(* IEC 61131-3 sources: Yaha/Documentation/Infomaterial/OSCAT/pcworx_basic_333/module_export (part 8) *)

(* ---- MS_TO_KMH.ST ---- *)
(*@PROPERTIES_EX@
TYPE: POU
LOCALE: 0
IEC_LANGUAGE: ST
PLC_TYPE: independent
PROC_TYPE: independent
GROUP: ENGINEERING.CONVERSION
*)
(*@KEY@:DESCRIPTION*)
version 1.0	4 Feb 2007
programmer 	hugo
tested by	tobias

this function converts velocities from Meters / Second to Kilometers / hour.
(*@KEY@:END_DESCRIPTION*)
FUNCTION MS_TO_KMH:REAL

(*Group:Default*)

VAR_INPUT
	MS :	REAL;
END_VAR

(*@KEY@: WORKSHEET
NAME: MS_TO_KMH
IEC_LANGUAGE: ST
*)
MS_TO_KMH := ms * 3.6;
(*@KEY@: END_WORKSHEET *)
END_FUNCTION

(* ---- MUL_ADD.ST ---- *)
(*@PROPERTIES_EX@
TYPE: POU
LOCALE: 0
IEC_LANGUAGE: ST
PLC_TYPE: independent
PROC_TYPE: independent
GROUP: MATHEMATICAL.MATHE
*)
(*@KEY@:DESCRIPTION*)
version 1.1	11 nov 2007
programmer 	hugo
tested by	tobias

this function multiplies an input X with K and adds Offset O to the result.
(*@KEY@:END_DESCRIPTION*)
FUNCTION MUL_ADD:REAL

(*Group:Default*)

VAR_INPUT
	X :	REAL;
	K :	REAL;
	O :	REAL;
END_VAR

(*@KEY@: WORKSHEET
NAME: MUL_ADD
IEC_LANGUAGE: ST
*)
MUL_ADD := X * K + O;
(*@KEY@: END_WORKSHEET *)
END_FUNCTION

(* ---- MULTI_IN.ST ---- *)
(*@PROPERTIES_EX@
TYPE: POU
LOCALE: 0
IEC_LANGUAGE: ST
PLC_TYPE: independent
PROC_TYPE: independent
GROUP: ENGINEERING.SENSOR
*)
(*@KEY@:DESCRIPTION*)
version 1.4	18. jul. 2009
programmer 	oscat
tested by	oscat

multi_in is a signal conditioning function which can be configured in 8 different ways.
it is used to read multiple sensors for the same value and protect the user from broken sensors or invalid data from sensors.

multi_in can be configured in different ways:
	mode = 0 means the the avg of the 3 inputs is used, this mode is the default mode.
	mode = 1 means in_1 is used.
	mode = 2 means in_2 is used.
	mode = 3 means in_3 is used.
	mode = 4 means default is used.
	mode = 5 means the lowest of the 3 external temperatures is used.
	mode = 6 means the higest externnal temperature is used.
	mode = 7 means the midlle input is used, if there are only two working, the lowest input is used.
	mode > 7 ,eans output is 0 at all times.
	in any config mode, an input higher then in_max or lower then in_min is ignored to prevent values from broken sensors or wires.
	if all inputs are higher then in_max or lower then in_min, a default value (default) is used.

(*@KEY@:END_DESCRIPTION*)
FUNCTION MULTI_IN:REAL

(*Group:Default*)

VAR_INPUT
	IN_1 :	REAL;
	IN_2 :	REAL;
	IN_3 :	REAL;
	DEFAULT :	REAL;
	IN_MIN :	REAL;
	IN_MAX :	REAL;
	MODE :	BYTE;
END_VAR

VAR
	count :	INT;
	F1 :	BOOL;
	F2 :	BOOL;
	F3 :	BOOL;
END_VAR

(*@KEY@: WORKSHEET
NAME: MULTI_IN
IEC_LANGUAGE: ST
*)
F1 :=  in_1 > in_min AND in_1 < in_max;
F2 :=  in_2 > in_min AND in_2 < in_max;
F3 :=  in_3 > in_min AND in_3 < in_max;

CASE _BYTE_TO_INT(mode) OF
0:	count := 0;
	IF F1 THEN
		count := count + 1;
		MULTI_IN := in_1;
	ELSE
		MULTI_IN := 0.0;
	END_IF;
	IF F2 THEN
		count := count + 1;
		MULTI_IN := MULTI_IN + in_2;
	END_IF;
	IF F3 THEN
		count := count + 1;
		MULTI_IN := MULTI_IN + in_3;
	END_IF;
	MULTI_IN := SEL_REAL(count = 0, MULTI_IN / INT_TO_REAL(count), default);

1:	MULTI_IN := SEL_REAL(F1, default, IN_1);

2:	MULTI_IN := SEL_REAL(F2, default, IN_2);

3:	MULTI_IN := SEL_REAL(F3, default, IN_3);

4:	MULTI_IN := default;

5:	MULTI_IN := SEL_REAL(F1, in_max, IN_1);
	IF F2 AND in_2 < MULTI_IN THEN MULTI_IN := in_2; END_IF;
	IF F3 AND in_3 < MULTI_IN THEN MULTI_IN := in_3; END_IF;
	IF MULTI_IN = in_max THEN MULTI_IN := default; END_IF;

6:	MULTI_IN := SEL_REAL(F1, in_min, IN_1);
	IF F2 AND in_2 > MULTI_IN THEN MULTI_IN := in_2; END_IF;
	IF F3 AND in_3 > MULTI_IN THEN MULTI_IN := in_3; END_IF;
	IF MULTI_IN = in_min THEN MULTI_IN := default; END_IF;

7:	IF F1 AND F2 AND F3 THEN MULTI_IN := MID3(in_1, in_2, in_3);
	ELSIF F1 AND F2 THEN MULTI_IN := MIN(in_1, in_2);
	ELSIF F1 AND F3 THEN MULTI_IN := MIN(in_1, in_3);
	ELSIF F2 AND F3 THEN MULTI_IN := MIN(in_2, in_3);
	ELSIF F1 THEN MULTI_IN := in_1;
	ELSIF F2 THEN MULTI_IN := in_2;
	ELSIF F3 THEN MULTI_IN := in_3;
	ELSE MULTI_IN := default;
	END_IF;

END_CASE;

(*
hm 1.1.2007		rev 1.1
	changed midr to mid3 function

hm	14. 10. 2008	rev 1.2
	corrected an error for in_3 overrange detection
	improved performance

hm	11. mar. 2009	rev 1.3
	changed real constants to use dot syntax

hm	18. jul. 2009	rev 1.4
	improved performance
*)

(*@KEY@: END_WORKSHEET *)
END_FUNCTION

(* ---- MULTIME.ST ---- *)
(*@PROPERTIES_EX@
TYPE: POU
LOCALE: 0
IEC_LANGUAGE: ST
PLC_TYPE: independent
PROC_TYPE: independent
GROUP: TIME_DATE
*)
(*@KEY@:DESCRIPTION*)
version 1.1	14 mar 2008
programmer 	hugo
tested by	tobias

multiplies a time by a real number and returns a time
(*@KEY@:END_DESCRIPTION*)
FUNCTION MULTIME:TIME

(*Group:Default*)

VAR_INPUT
	T :	TIME;
	M :	REAL;
END_VAR

(*@KEY@: WORKSHEET
NAME: MULTIME
IEC_LANGUAGE: ST
*)
multime := DWORD_TO_TIME(_REAL_TO_DWORD(_DWORD_TO_REAL(TIME_TO_DWORD(t))*M));

(* revision history
hm		2. oct 2006	rev 1.0
	original version

hm		14. mar 2008	rev 1.1
	rounded the result after the last digit

*)
(*@KEY@: END_WORKSHEET *)
END_FUNCTION

(* ---- MUX_2.ST ---- *)
(*@PROPERTIES_EX@
TYPE: POU
LOCALE: 0
IEC_LANGUAGE: ST
PLC_TYPE: independent
PROC_TYPE: independent
GROUP: LOGIC.GATE_LOGIC
*)
(*@KEY@:DESCRIPTION*)
version 1.2	16. oct. 2008
programmer 	hugo
tested BY	oscat

dual input multiplexer
depending on the value of A0, D0 or D1 will be switched to the Output
(*@KEY@:END_DESCRIPTION*)
FUNCTION MUX_2:BOOL

(*Group:Default*)

VAR_INPUT
	D0 :	BOOL;
	D1 :	BOOL;
	A0 :	BOOL;
END_VAR

(*@KEY@: WORKSHEET
NAME: MUX_2
IEC_LANGUAGE: ST
*)
MUX_2 := SEL(A0, D0, D1);

(*
revision history:
hm	5.10.2006		rev 1.1
	changed to ST Langage for better portability.

hm	16. oct. 2008	rev 1.2
	improved performance

*)
(*@KEY@: END_WORKSHEET *)
END_FUNCTION

(* ---- MUX_4.ST ---- *)
(*@PROPERTIES_EX@
TYPE: POU
LOCALE: 0
IEC_LANGUAGE: ST
PLC_TYPE: independent
PROC_TYPE: independent
GROUP: LOGIC.GATE_LOGIC
*)
(*@KEY@:DESCRIPTION*)
version 1.2	16. oct. 2008
programmer 	hugo
tested BY	oscat

quad input multiplexer
depending on the value of A0 and A1, one of the 4 inputs will be switched to the Output
(*@KEY@:END_DESCRIPTION*)
FUNCTION MUX_4:BOOL

(*Group:Default*)

VAR_INPUT
	D0 :	BOOL;
	D1 :	BOOL;
	D2 :	BOOL;
	D3 :	BOOL;
	A0 :	BOOL;
	A1 :	BOOL;
END_VAR

(*@KEY@: WORKSHEET
NAME: MUX_4
IEC_LANGUAGE: ST
*)
IF A1 THEN
	MUX_4 := SEL(A0, D2, D3);
ELSE
	MUX_4 := SEL(A0, D0, D1);
END_IF;

(*
revision history:
hm 	5.10.2006		rev 1.1
	rewritten to ST for better portability

hm	16. oct. 2008	rev 1.2
	improved performance

*)
(*@KEY@: END_WORKSHEET *)
END_FUNCTION

(* ---- MUX_R2.ST ---- *)
(*@PROPERTIES_EX@
TYPE: POU
LOCALE: 0
IEC_LANGUAGE: ST
PLC_TYPE: independent
PROC_TYPE: independent
GROUP: ENGINEERING.SIGNAL_PROCESSING
*)
(*@KEY@:DESCRIPTION*)
version 1.1	16. oct. 2008
programmer 	oscat
tested by	oscat

MUX_R2 is an analog Multiplexer.
one of 2 real inputs are selected and put through to out.
The Adress input A selects between 2 Real inputs IN0 and IN1, A=0 > In0, A=1 > in1.
(*@KEY@:END_DESCRIPTION*)
FUNCTION MUX_R2:REAL

(*Group:Default*)

VAR_INPUT
	IN0 :	REAL;
	IN1 :	REAL;
	A :	BOOL;
END_VAR

(*@KEY@: WORKSHEET
NAME: MUX_R2
IEC_LANGUAGE: ST
*)
MUX_R2 := SEL(A, IN0, IN1);

(* revision history
hm	19. jan. 2007	rev 1.0
	original version

hm	16. oct. 2008	rev 1.1
	improved performance
*)
(*@KEY@: END_WORKSHEET *)
END_FUNCTION

(* ---- MUX_R4.ST ---- *)
(*@PROPERTIES_EX@
TYPE: POU
LOCALE: 0
IEC_LANGUAGE: ST
PLC_TYPE: independent
PROC_TYPE: independent
GROUP: ENGINEERING.SIGNAL_PROCESSING
*)
(*@KEY@:DESCRIPTION*)
version 1.1	16. oct. 2008
programmer 	oscat
tested by	oscat

MUX_R4 is an analog Multiplexer.
one of 4 real inputs are selected and put through to out.
The Adress input A0 and A1 selects between the 4 Real inputs IN0.. IN1.
(*@KEY@:END_DESCRIPTION*)
FUNCTION MUX_R4:REAL

(*Group:Default*)

VAR_INPUT
	IN0 :	REAL;
	IN1 :	REAL;
	IN2 :	REAL;
	IN3 :	REAL;
	A0 :	BOOL;
	A1 :	BOOL;
END_VAR

(*@KEY@: WORKSHEET
NAME: MUX_R4
IEC_LANGUAGE: ST
*)
IF A1 THEN
	MUX_R4 := SEL(A0, IN2, IN3);
ELSE
	MUX_R4 := SEL(A0, IN0, IN1);
END_IF;

(* revision history
hm	19. jan 2007	rev 1.0
	original version

hm	16. oct. 2008	rev 1.1
	improved performance
*)
(*@KEY@: END_WORKSHEET *)
END_FUNCTION

(* ---- NEGX.ST ---- *)
(*@PROPERTIES_EX@
TYPE: POU
LOCALE: 0
IEC_LANGUAGE: ST
PLC_TYPE: independent
PROC_TYPE: independent
GROUP: MATHEMATICAL.MATHE
*)
(*@KEY@:DESCRIPTION*)
version 1.0	26. oct. 2008
programmer 	hugo
tested by	tobias

This function returns -X
(*@KEY@:END_DESCRIPTION*)
FUNCTION NEGX:REAL

(*Group:Default*)

VAR_INPUT
	X :	REAL;
END_VAR

(*@KEY@: WORKSHEET
NAME: NEGX
IEC_LANGUAGE: ST
*)
NEGX := -X;

(* revision history
hm	26. oct. 2008	rev 1.0
	original version

*)
(*@KEY@: END_WORKSHEET *)
END_FUNCTION

(* ---- OFFSET.ST ---- *)
(*@PROPERTIES_EX@
TYPE: POU
LOCALE: 0
IEC_LANGUAGE: ST
PLC_TYPE: independent
PROC_TYPE: independent
GROUP: ENGINEERING.SIGNAL_PROCESSING
*)
(*@KEY@:DESCRIPTION*)
version 1.0	12 jan 2007
programmer 	oscat
tested by	tobias

The Function offset adds offsets to an analog signal depending on digital inputs.
all selected offsets are added at the same time.
with the input D a default value instead of the input X can be used.
(*@KEY@:END_DESCRIPTION*)
FUNCTION OFFSET:REAL

(*Group:Default*)

VAR_INPUT
	X :	REAL;
	O1 :	BOOL;
	O2 :	BOOL;
	O3 :	BOOL;
	O4 :	BOOL;
	D :	BOOL;
	OFFSET_1 :	REAL;
	OFFSET_2 :	REAL;
	OFFSET_3 :	REAL;
	OFFSET_4 :	REAL;
	DEFAULT :	REAL;
END_VAR

(*@KEY@: WORKSHEET
NAME: OFFSET
IEC_LANGUAGE: ST
*)
IF D THEN Offset := default; ELSE Offset := X; END_IF;
IF O1 THEN Offset := Offset + offset_1; END_IF;
IF O2 THEN Offset := Offset + offset_2; END_IF;
IF O3 THEN Offset := Offset + offset_3; END_IF;
IF O4 THEN Offset := Offset + offset_4; END_IF;
(*@KEY@: END_WORKSHEET *)
END_FUNCTION

(* ---- OFFSET2.ST ---- *)
(*@PROPERTIES_EX@
TYPE: POU
LOCALE: 0
IEC_LANGUAGE: ST
PLC_TYPE: independent
PROC_TYPE: independent
GROUP: ENGINEERING.SIGNAL_PROCESSING
*)
(*@KEY@:DESCRIPTION*)
version 1.0	12 jan 2007
programmer 	oscat
tested by	tobias

The Function offset adds offsets to an analog signal depending on digital inputs.
one offset can be added at the same time, if more then one input is true, the one with the highest number (o1 .. o4) will be used.
The input D will select a default value instead of X for input.
(*@KEY@:END_DESCRIPTION*)
FUNCTION OFFSET2:REAL

(*Group:Default*)

VAR_INPUT
	X :	REAL;
	O1 :	BOOL;
	O2 :	BOOL;
	O3 :	BOOL;
	O4 :	BOOL;
	D :	BOOL;
	OFFSET_1 :	REAL;
	OFFSET_2 :	REAL;
	OFFSET_3 :	REAL;
	OFFSET_4 :	REAL;
	DEFAULT :	REAL;
END_VAR

(*@KEY@: WORKSHEET
NAME: OFFSET2
IEC_LANGUAGE: ST
*)
IF D THEN Offset2 := default; ELSE Offset2 := X; END_IF;
IF O4 THEN Offset2 := Offset2 + offset_4;
ELSIF O3 THEN Offset2 := Offset2 + offset_3;
ELSIF O2 THEN Offset2 := Offset2 + offset_2;
ELSIF O1 THEN Offset2 := Offset2 + offset_1;
END_IF;
(*@KEY@: END_WORKSHEET *)
END_FUNCTION

(* ---- OM_TO_F.ST ---- *)
(*@PROPERTIES_EX@
TYPE: POU
LOCALE: 0
IEC_LANGUAGE: ST
PLC_TYPE: independent
PROC_TYPE: independent
GROUP: ENGINEERING.CONVERSION
*)
(*@KEY@:DESCRIPTION*)
version 1.1	18. oct. 2008
programmer 	hugo
tested by		tobias

this function converts Omega F to frequency
F = OM / (2*PI)
(*@KEY@:END_DESCRIPTION*)
FUNCTION OM_TO_F:REAL

(*Group:Default*)

VAR_INPUT
	OM :	REAL;
END_VAR

(*@KEY@: WORKSHEET
NAME: OM_TO_F
IEC_LANGUAGE: ST
*)
OM_to_F := OM / 6.283185307179586476;

(* revision history
hm	22. jan. 2007	rev 1.0
	original version

hm	18. oct. 2008	rev 1.1
	using math constants

*)
(*@KEY@: END_WORKSHEET *)
END_FUNCTION

(* ---- OSCAT_VERSION.ST ---- *)
(*@PROPERTIES_EX@
TYPE: POU
LOCALE: 0
IEC_LANGUAGE: ST
PLC_TYPE: independent
PROC_TYPE: independent
GROUP: OTHER
*)
(*@KEY@:DESCRIPTION*)
version 1.1	16 dec 2007
programmer 	hugo
tested by	tobias

oscat_version returns the version number in dword format
132 is library version 1.32
if IN = true, the release date will be returned
(*@KEY@:END_DESCRIPTION*)
FUNCTION OSCAT_VERSION:DWORD

(*Group:Default*)

VAR_INPUT
	IN :	BOOL;
END_VAR

(*@KEY@: WORKSHEET
NAME: OSCAT_VERSION
IEC_LANGUAGE: ST
*)
IF in THEN
	Oscat_version := UDINT_TO_DWORD(set_Date(2012,01,02));
ELSE
	Oscat_version := DWORD#333;
END_IF;

(* revision history
hm	6. oct 2006	rev 1.0
	original version

hm	16. dec 2007	rev 1.1
	added possibility to return date and version depending on IN.

*)
(*@KEY@: END_WORKSHEET *)
END_FUNCTION

(* ---- PARITY.ST ---- *)
(*@PROPERTIES_EX@
TYPE: POU
LOCALE: 0
IEC_LANGUAGE: ST
PLC_TYPE: independent
PROC_TYPE: independent
GROUP: LOGIC.GATE_LOGIC
*)
(*@KEY@:DESCRIPTION*)
version 1.3	18 feb 2008
programmer 	hugo
tested BY	hans

this function calculates the even parity of an input Dword
the output will be true if the amount of high bits are an odd number.
(*@KEY@:END_DESCRIPTION*)
FUNCTION PARITY:BOOL

(*Group:Default*)

VAR_INPUT
	IN :	DWORD;
END_VAR

VAR
	in2 :	DWORD;
END_VAR

(*@KEY@: WORKSHEET
NAME: PARITY
IEC_LANGUAGE: ST
*)
in2:=in;
WHILE in2 > DWORD#0 DO
	parity := parity XOR BIT_OF_DWORD(in2,0) XOR BIT_OF_DWORD(in2,1) XOR BIT_OF_DWORD(in2,2) XOR BIT_OF_DWORD(in2,3);
	in2 := SHR(in2,4);
END_WHILE;

(* code before rev 1.2
WHILE in > 0 DO
	IF in.0 THEN cnt := cnt +1; END_IF;
	in := SHR(in,1);
END_WHILE;
IF (cnt MOD 2) = 1 THEN parity := TRUE; ELSE parity := FALSE; END_IF;
*)

(* revision history

rev 1.0 hm 1 sep 2006
	original version

rev 1.1 hm 10.9.2007
	changed algorithm to improve performance

rev 1.2	hm	8 dec 2007
	changed algorithm to improve performance

rev 1.3	hm	18 feb 2008
	changed algorithm to improve performance
*)
(*@KEY@: END_WORKSHEET *)
END_FUNCTION

(* ---- PERIOD.ST ---- *)
(*@PROPERTIES_EX@
TYPE: POU
LOCALE: 0
IEC_LANGUAGE: ST
PLC_TYPE: independent
PROC_TYPE: independent
GROUP: TIME_DATE
*)
(*@KEY@:DESCRIPTION*)
version 1.3	22. mar. 2008
programmer 	hugo
tested by	tobias

PERIOD checks if a given date is between two dates (d1 and d2) d1 is the starting date and d2 the last date for the period.
the years of the dates are ignored, so the function period cheks for a time period within a year independet of the year.
(*@KEY@:END_DESCRIPTION*)
FUNCTION PERIOD:BOOL

(*Group:Default*)

VAR
	day1 :	INT;
	day2 :	INT;
	dayx :	INT;
END_VAR

VAR_INPUT
	D1 :	UDINT;
	Dx :	UDINT;
	D2 :	UDINT;
END_VAR

(*@KEY@: WORKSHEET
NAME: PERIOD
IEC_LANGUAGE: ST
*)
day1 := day_of_year(d1);
day2 := day_of_year(d2);
dayx := day_of_year(dx);
IF NOT leap_of_Date(dx) AND dayx > 58 THEN dayx := dayx + 1; END_IF;
IF NOT leap_of_Date(d1) AND day1 > 58 THEN day1 := day1 + 1; END_IF;
IF NOT leap_of_Date(d2) AND day2 > 58 THEN day2 := day2 + 1; END_IF;

IF day2 < day1 THEN
	(* the period spans over the new year *)
	period := dayx <= day2 OR dayx >= day1;
ELSE
	period := dayx >= day1 AND dayx <= day2;
END_IF;

(* code before rev 1.2
yx := year(dx);
p1 := date_add(d1,0,0,0,yx - year(d1));
p2 := date_add(d2,0,0,0,yx - year(d2));

IF p2 >= p1 THEN
	period := dx <= p2  AND dx >= p1;
ELSE
	period := dx <= p2 OR dx >= p1;
END_IF;
*)

(* revision history

hm		19. sep 2007	rev 1.0
	original version

hm		20. sep 2007	rev 1.1
	corrected a problem with leap year

hm		4. jan 2008		rev 1.2
	changed code for better performance

hm		22. mar. 2008	rev 1.3
	function would deliver wrong results when d1, d2 or dx are a leap_year

*)
(*@KEY@: END_WORKSHEET *)
END_FUNCTION

(* ---- PT_TO_F.ST ---- *)
(*@PROPERTIES_EX@
TYPE: POU
LOCALE: 0
IEC_LANGUAGE: ST
PLC_TYPE: independent
PROC_TYPE: independent
GROUP: ENGINEERING.CONVERSION
*)
(*@KEY@:DESCRIPTION*)
version 1.1	11. mar. 2009
programmer 	hugo
tested by	tobias

this function converts periode time to frequency
(*@KEY@:END_DESCRIPTION*)
FUNCTION PT_TO_F:REAL

(*Group:Default*)

VAR_INPUT
	PT :	TIME;
END_VAR

(*@KEY@: WORKSHEET
NAME: PT_TO_F
IEC_LANGUAGE: ST
*)
PT_TO_F := 1000.0 / _DWORD_TO_REAL(TIME_TO_DWORD(PT));

(*	revision history
hm	4. aug. 2006	rev 1.0
	original version

hm	11. mar. 2009	rev 1.1
	real constants updated to new systax using dot

*)
(*@KEY@: END_WORKSHEET *)
END_FUNCTION

(* ---- RAD.ST ---- *)
(*@PROPERTIES_EX@
TYPE: POU
LOCALE: 0
IEC_LANGUAGE: ST
PLC_TYPE: independent
PROC_TYPE: independent
GROUP: MATHEMATICAL.MATHE
*)
(*@KEY@:DESCRIPTION*)
version 1.2	18. oct. 2008
programmer 	hugo
tested by	tobias

this function converts Radiant to degrees
(*@KEY@:END_DESCRIPTION*)
FUNCTION RAD:REAL

(*Group:Default*)

VAR_INPUT
	DEG :	REAL;
END_VAR

(*@KEY@: WORKSHEET
NAME: RAD
IEC_LANGUAGE: ST
*)
Rad := modR(0.0174532925199433 * deg , 6.283185307179586476);

(* revision history
hm	4. aug 2006		rev 1.0
	original version

hm 	16. oct 2007	rev 1.1
	added modr statement which prohibits rad to become bigger than 2PI

hm	18. oct 2008	rev 1.2
	using math constants

*)
(*@KEY@: END_WORKSHEET *)
END_FUNCTION

(* ---- RANGE_TO_BYTE.ST ---- *)
(*@PROPERTIES_EX@
TYPE: POU
LOCALE: 0
IEC_LANGUAGE: ST
PLC_TYPE: independent
PROC_TYPE: independent
GROUP: ENGINEERING.SIGNAL_PROCESSING
*)
(*@KEY@:DESCRIPTION*)
version 1.0	9. jan 2008
programmer 	hugo
tested by		tobias

Range_to_byte converts a real value between low and high into a byte
(*@KEY@:END_DESCRIPTION*)
FUNCTION RANGE_TO_BYTE:BYTE

(*Group:Default*)

VAR_INPUT
	X :	REAL;
	LOW :	REAL;
	HIGH :	REAL;
END_VAR

(*@KEY@: WORKSHEET
NAME: RANGE_TO_BYTE
IEC_LANGUAGE: ST
*)
Range_to_Byte := REAL_TO_BYTE(TRUNC_REAL((LIMIT(low,X,high)-low) * 255.0 / (high - low)));

(* revision history
hm	9. jan 2008		rev 1.0
	original version

*)
(*@KEY@: END_WORKSHEET *)
END_FUNCTION

(* ---- RANGE_TO_WORD.ST ---- *)
(*@PROPERTIES_EX@
TYPE: POU
LOCALE: 0
IEC_LANGUAGE: ST
PLC_TYPE: independent
PROC_TYPE: independent
GROUP: ENGINEERING.SIGNAL_PROCESSING
*)
(*@KEY@:DESCRIPTION*)
version 1.0	9. jan 2008
programmer 	hugo
tested by	tobias

Range_to_word converts a real value between low and high into a byte
(*@KEY@:END_DESCRIPTION*)
FUNCTION RANGE_TO_WORD:WORD

(*Group:Default*)

VAR_INPUT
	X :	REAL;
	LOW :	REAL;
	HIGH :	REAL;
END_VAR

(*@KEY@: WORKSHEET
NAME: RANGE_TO_WORD
IEC_LANGUAGE: ST
*)
Range_to_Word := REAL_TO_WORD(TRUNC_REAL((LIMIT(low,X,high)-low) * 65535.0 / (high - low)));

(* revision history
hm	9. jan 2008		rev 1.0
	original version

*)
(*@KEY@: END_WORKSHEET *)
END_FUNCTION

(* ---- REFLECT.ST ---- *)
(*@PROPERTIES_EX@
TYPE: POU
LOCALE: 0
IEC_LANGUAGE: ST
PLC_TYPE: independent
PROC_TYPE: independent
GROUP: LOGIC.GATE_LOGIC
*)
(*@KEY@:DESCRIPTION*)
version 1.0	16. jan 2011
programmer 	hugo
tested BY	tobias

This function reverses the specified amount of bits from bit 0 to bit n within a dword  while L specifies the amount of Bits to be reflected.

(*@KEY@:END_DESCRIPTION*)
FUNCTION REFLECT:DWORD

(*Group:Default*)

VAR_INPUT
	D :	DWORD;
	L :	INT;
END_VAR

VAR
	i :	INT;
	_d :	DWORD;
END_VAR

(*@KEY@: WORKSHEET
NAME: REFLECT
IEC_LANGUAGE: ST
*)
REFLECT := DWORD#0;
_d := D;
FOR i := 1 TO L DO
	REFLECT := SHL(REFLECT, 1) OR BOOL_TO_DWORD((_d AND DWORD#2#0000_0001) > DWORD#0); (* D.0 *)
	_d := SHR(_d, 1);
END_FOR;
REFLECT := REFLECT OR SHL(_d, L);

(* revision history
hm	 16. jan 2011
	new module

*)
(*@KEY@: END_WORKSHEET *)
END_FUNCTION

(* ---- REFRACTION.ST ---- *)
(*@PROPERTIES_EX@
TYPE: POU
LOCALE: 0
IEC_LANGUAGE: ST
PLC_TYPE: independent
PROC_TYPE: independent
GROUP: TIME_DATE
*)
(*@KEY@:DESCRIPTION*)
version 1.1	7. mar. 2009
programmer 	hugo
tested by	oscat

REFRACTION calculates the atmospheric refraction in degrees.
the input angle goes from 0 at the hirizon to 90 at midday.
(*@KEY@:END_DESCRIPTION*)
FUNCTION REFRACTION:REAL

(*Group:Default*)

VAR_INPUT
	ELEV :	REAL;
END_VAR

VAR
	tmp :	REAL;
END_VAR

(*@KEY@: WORKSHEET
NAME: REFRACTION
IEC_LANGUAGE: ST
*)
tmp := LIMIT(-1.9, elev, 80.0);
REFRACTION := 0.0174532925199433 / TAN(0.0174532925199433 * (tmp + 10.3 / (tmp + 5.11)));

(* revision histroy
hm	14. jul. 2008	rev 1.0
	original release

hm	7. mar. 2009	rev 1.1
	using new formula

*)

(*@KEY@: END_WORKSHEET *)
END_FUNCTION

(* ---- RES_NI.ST ---- *)
(*@PROPERTIES_EX@
TYPE: POU
LOCALE: 0
IEC_LANGUAGE: ST
PLC_TYPE: independent
PROC_TYPE: independent
GROUP: ENGINEERING.SENSOR
*)
(*@KEY@:DESCRIPTION*)
version 1.2	2 dec 2007
programmer 	hugo
tested by	tobias

this function returs the resistance for a nickel sensor for a temperature range from -60..+180 °C *)
(*@KEY@:END_DESCRIPTION*)
FUNCTION RES_NI:REAL

(*Group:Default*)

VAR_INPUT
	T :	REAL;
	R0 :	REAL;
END_VAR

VAR
	T2 :	REAL;
END_VAR

(*@KEY@: WORKSHEET
NAME: RES_NI
IEC_LANGUAGE: ST
*)
T2 := T*T;
Res_NI := R0 + 0.5485*T + 0.665E-3*T2 + 2.805E-9*T2*T2;

(* revision history

hm	4.8.2006		rev 1.0
	original version

hm	13.9.2007		rev 1.1
	changed coding for better performance

hm	2. dec. 2007	rev 1.2
	changed code for better performance
*)

(*

 Auszug aus DIN 43760 für Ni100

°C		R		°C		R		°C	R		°C		R		°C		R

-60 	69,5 	-10 	94,6 	40 	123,0 	90 		154,9 	140 	190,9
-55 	71,9 	-5 		97,3 	45 	126,0 	95 		158,3 	145 	194,8
-50 	74,3 	0 		100,0 	50 	129,1 	100 	161,8 	150 	198,7
-45 	76,7 	5 		102,8 	55 	132,2 	105 	165,3 	155 	202,6
-40 	79,1 	10 		105,6 	60 	135,3 	110 	168,8 	160 	206,6
-35 	81,6 	15 		108,4 	65 	138,5 	115 	172,4 	165 	210,7
-30 	84,2 	20 		111,2 	70 	141,7 	120 	176,0 	170 	214,8
-25 	86,7 	25 		114,1 	75 	145,0 	125 	179,6 	175 	219,0
-20 	89,3 	30 		117,1 	80 	148,3 	130 	183,3 	180 	223,2
-15 	91,9 	35 		120,0 	85 	151,6 	135 	187,1

*)
(*@KEY@: END_WORKSHEET *)
END_FUNCTION

(* ---- RES_NTC.ST ---- *)
(*@PROPERTIES_EX@
TYPE: POU
LOCALE: 0
IEC_LANGUAGE: ST
PLC_TYPE: independent
PROC_TYPE: independent
GROUP: ENGINEERING.SENSOR
*)
(*@KEY@:DESCRIPTION*)
version 1.1	11. mar. 2009
programmer 	hugo
tested by	tobias

this function returs the resistance for a NTC sensor for a given temperature in °C.
RN is the resistance at 25 °C and B is a constant for the given sensor.

(*@KEY@:END_DESCRIPTION*)
FUNCTION RES_NTC:REAL

(*Group:Default*)

VAR_INPUT
	T :	REAL;
	RN :	REAL;
	B :	REAL;
END_VAR

(*@KEY@: WORKSHEET
NAME: RES_NTC
IEC_LANGUAGE: ST
*)
RES_NTC := RN * EXP(B * (1.0 / (T+273.15) - 0.00335401643468053));

(* revision history

hm 30. dec. 2008	rev 1.0
	original version

hm	11. mar. 2009	rev 1.1
	changed real constants to use dot syntax

*)
(*@KEY@: END_WORKSHEET *)
END_FUNCTION

(* ---- RES_PT.ST ---- *)
(*@PROPERTIES_EX@
TYPE: POU
LOCALE: 0
IEC_LANGUAGE: ST
PLC_TYPE: independent
PROC_TYPE: independent
GROUP: ENGINEERING.SENSOR
*)
(*@KEY@:DESCRIPTION*)
version 1.3	11. mar. 2009
programmer 	hugo
tested by	oscat

this function returs the resistance for a platinum sensor for a temperature range from -200..+850 °C

(*@KEY@:END_DESCRIPTION*)
FUNCTION RES_PT:REAL

(*Group:Default*)

VAR_INPUT
	T :	REAL;
	R0 :	REAL;
END_VAR

VAR
	T2 :	REAL;
END_VAR

(*@KEY@: WORKSHEET
NAME: RES_PT
IEC_LANGUAGE: ST
*)
T2 := T * T;

IF T >= 0.0 THEN
	RES_PT := R0 * ( 1.0 + 3.90802E-3 * T + -5.802E-7 * T2);
ELSE
	RES_PT := R0 * ( 1.0 + 3.90802E-3 * T + -5.802E-7 * T2 + -4.27350E-12 * (T - 100.0) * T2 * T);
END_IF;

(* revision history
hm	4. aug. 2006	rev 1.1
	original version

hm	2. dec 2007	rev 1.2
	changed code for better performance

hm	11. mar. 2009	rev 1.3
	changed real constants to use dot syntax

*)

(*
 Auszug aus DIN 43760 für Pt100

°C		R		°C		R		°C	R			°C		R			°C		R			°C		R

-200 	18,49 	-100 	60,25 	0 	100,00 	100 	138,50 	200 	175,84 	300 	212,02
-195 	20,65 	-95 	62,28 	5 	101,95 	105 	140,39 	205 	177,68 	305 	213,80
-190 	22,80 	-90 	64,30 	10 	103,90 	110 	142,29 	210 	179,51 	310 	215,57
-185 	24,94 	-85 	66,31 	15 	105,85 	115 	144,17 	215 	181,34 	315 	217,35
-180 	27,08 	-80 	68,33 	20 	107,79 	120 	146,06 	220 	183,17 	320 	219,12
-175 	29,20 	-75 	70,33 	25 	109,73 	125 	147,94 	225 	184,99 	325 	220,88
-170 	31,32 	-70 	72,33 	30 	111,67 	130 	149,82 	230 	186,82 	330 	222,65
-165 	33,43 	-65 	74,33 	35 	113,61 	135 	151,70 	235 	188,63 	335 	224,41
-160 	35,33 	-60 	76,33 	40 	115,54 	140 	153,58 	240 	190,45 	340 	226,17
-155 	37,63 	-55 	78,32 	45 	117,47 	145 	155,45 	245 	192,26 	345 	227,92
-150 	39,71 	-50 	80,31 	50 	119,40 	150 	157,31 	250 	194,07 	350 	229,67
-145 	41,79 	-45 	82,29 	55 	121,32 	155 	159,18 	255 	195,88 	355 	231,42
-140 	43,87 	-40 	84,27 	60 	123,24 	160 	161,04 	260 	197,69 	360 	233,17
-135 	45,94 	-35 	86,25 	65 	125,16 	165 	162,90 	265 	199,49 	365 	234,91
-130 	48,00 	-30 	88,22 	70 	127,07 	170 	164,76 	270 	201,29 	370 	236,65
-125 	50,06 	-25 	90,19 	75 	128,98 	175 	166,61 	275 	203,08 	375 	238,39
-120 	52,11 	-20 	92,16 	80 	130,89 	180 	168,46 	280 	204,88 	380 	240,13
-115 	54,15 	-15 	94,12 	85 	132,80 	185 	170,31 	285 	206,67 	385 	241,86
-110 	56,19 	-10 	96,09 	90 	134,70 	190 	172,16 	290 	208,45 	390 	243,59
-105 	58,22 	-5 		98,04 	95 	136,60 	195 	174,00 	295 	210,24 	395 	245,31

*)
(*
revision history

*)
(*@KEY@: END_WORKSHEET *)
END_FUNCTION

(* ---- RES_SI.ST ---- *)
(*@PROPERTIES_EX@
TYPE: POU
LOCALE: 0
IEC_LANGUAGE: ST
PLC_TYPE: independent
PROC_TYPE: independent
GROUP: ENGINEERING.SENSOR
*)
(*@KEY@:DESCRIPTION*)
version 1.2	11. mar. 2009
programmer 	hugo
tested by	tobias

this function returs the resistance for a silicon sensor for a temperature range from -50..+150 °C
for example KTY10 normaly Rs at 25 °C
(*@KEY@:END_DESCRIPTION*)
FUNCTION RES_SI:REAL

(*Group:Default*)

VAR_INPUT
	T :	REAL;
	RS :	REAL;
	TS :	REAL;
END_VAR

VAR
	TX :	REAL;
END_VAR

(*@KEY@: WORKSHEET
NAME: RES_SI
IEC_LANGUAGE: ST
*)
TX := T - TS;
RES_SI := RS * ( 1.0 + 7.64E-3 * TX + 1.66E-5 * TX * TX);

(* revision history
hm	4. aug 2006	rev 1.0
	original version

hm	2. dec 2007	rev 1.1
	changed code for better performance

hm	11. mar. 2009	rev 1.2
	changed real constants to use dot syntax

*)
(*@KEY@: END_WORKSHEET *)
END_FUNCTION

(* ---- REVERSE.ST ---- *)
(*@PROPERTIES_EX@
TYPE: POU
LOCALE: 0
IEC_LANGUAGE: ST
PLC_TYPE: independent
PROC_TYPE: independent
GROUP: LOGIC.GATE_LOGIC
*)
(*@KEY@:DESCRIPTION*)
version 1.1	18. feb 2008
programmer 	hugo
tested BY	tobias

This function reverses the bits of a byte so that after execution bit 7 is at bit 0 location and so forth.
(*@KEY@:END_DESCRIPTION*)
FUNCTION REVERSE:BYTE

(*Group:Default*)

VAR_INPUT
	IN :	BYTE;
END_VAR

(*@KEY@: WORKSHEET
NAME: REVERSE
IEC_LANGUAGE: ST
*)
reverse := SHL_BYTE(in,7) OR SHR_BYTE(in,7) OR (ROR_BYTE(in,3) AND BYTE#2#01000100) OR (ROL_BYTE(in,3) AND BYTE#2#00100010)
	OR (SHL_BYTE(in,1) AND BYTE#2#00010000) OR (SHR_BYTE(in,1) AND BYTE#2#00001000);

(* revision history
hm		9.oct 2007		rev 1.0
	original version

hm		18. feb 2008	rev 1.1
	improved performance
*)
(*@KEY@: END_WORKSHEET *)
END_FUNCTION

(* ---- RND.ST ---- *)
(*@PROPERTIES_EX@
TYPE: POU
LOCALE: 0
IEC_LANGUAGE: ST
PLC_TYPE: independent
PROC_TYPE: independent
GROUP: MATHEMATICAL.MATHE
*)
(*@KEY@:DESCRIPTION*)
version 1.2	10. mar. 2009
programmer 	hugo
tested by	tobias

this function rounds a real down to n digits total.
round(3.1415,2) = 3.1

(*@KEY@:END_DESCRIPTION*)
FUNCTION RND:REAL

(*Group:Default*)

VAR_INPUT
	X :	REAL;
	N :	INT;
END_VAR

VAR
	M :	REAL;
END_VAR

(*@KEY@: WORKSHEET
NAME: RND
IEC_LANGUAGE: ST
*)
IF X = 0.0 THEN
	RND := 0.0;
ELSE
	M := EXPN(10.0,N - CEIL(LOG(ABS(X))));
	RND := DINT_TO_REAL(_REAL_TO_DINT(X * M)) / M;
END_IF;

(* revision history
hm	11. mar 2008	rev 1.0
	original version

hm	26. oct. 2008	rev 1.1
	code optimization

hm	10. mar. 2009	rev 1.2
	real constants updated to new systax using dot

*)

(*@KEY@: END_WORKSHEET *)
END_FUNCTION

(* ---- ROUND.ST ---- *)
(*@PROPERTIES_EX@
TYPE: POU
LOCALE: 0
IEC_LANGUAGE: ST
PLC_TYPE: independent
PROC_TYPE: independent
GROUP: MATHEMATICAL.MATHE
*)
(*@KEY@:DESCRIPTION*)
version 1.4	16. mar 2008
programmer 	hugo
tested by	tobias

this function rounds a real down to n digits behind the comma.
round(3.1415,1) = 3.1
(*@KEY@:END_DESCRIPTION*)
FUNCTION ROUND:REAL

(*Group:Default*)

VAR_INPUT
	IN :	REAL;
	N :	INT;
END_VAR

VAR
	X :	REAL;
END_VAR

(*@KEY@: WORKSHEET
NAME: ROUND
IEC_LANGUAGE: ST
*)
IF N < 4 THEN
	IF N < 2 THEN
		IF N = 0 THEN X := 1.0; ELSE X := 10.0; END_IF;
	ELSE
		IF N = 2 THEN X := 100.0; ELSE X := 1000.0; END_IF;
	END_IF;
ELSE
	IF N < 6 THEN
		IF N = 4 THEN X := 10000.0; ELSE X := 100000.0; END_IF;
	ELSE
		IF N = 6 THEN X := 1000000.0; ELSE X := 10000000.0; END_IF;
	END_IF;
END_IF;

ROUND := DINT_TO_REAL(_REAL_TO_DINT(in * X)) / X;

(*
IF in >= 0 THEN
	ROUND := TRUNC(in * X + 0.5) / X;
ELSE
	ROUND := TRUNC(in * X - 0.5) / X;
END_IF;
*)

(* revision history
hm	1. sep 2006	rev 1.0
	original version

hm	2. dec 2007	rev 1.1
	changed code for better performance

hm	8. jan 2008	rev 1.2
	further improvement in performance

hm 11. mar. 2008	rev 1.3
	corrected an error with negative numbers
	use real_to_dint instead of trunc

hm	16. mar 2008	rev 1.4
	added type conversion to avoid warning under codesys 3.0
*)
(*@KEY@: END_WORKSHEET *)
END_FUNCTION

(* ---- SCALE.ST ---- *)
(*@PROPERTIES_EX@
TYPE: POU
LOCALE: 0
IEC_LANGUAGE: ST
PLC_TYPE: independent
PROC_TYPE: independent
GROUP: ENGINEERING.SIGNAL_PROCESSING
*)
(*@KEY@:DESCRIPTION*)
version 1.0	16. may. 2008
programmer 	hugo
tested by	tobias

Scale is used to translate an input x to output by the formula Y = X*K + O.
at the same time the output is limited to MN and MX.
(*@KEY@:END_DESCRIPTION*)
FUNCTION SCALE:REAL

(*Group:Default*)

VAR_INPUT
	X :	REAL;
	K :	REAL;
	O :	REAL;
	MX :	REAL;
	MN :	REAL;
END_VAR

(*@KEY@: WORKSHEET
NAME: SCALE
IEC_LANGUAGE: ST
*)
SCALE := LIMIT(MN, X * K + O, MX);

(* revision history
hm	16. may. 2008		rev 1.0
	original version
*)
(*@KEY@: END_WORKSHEET *)
END_FUNCTION

(* ---- SCALE_B.ST ---- *)
(*@PROPERTIES_EX@
TYPE: POU
LOCALE: 0
IEC_LANGUAGE: ST
PLC_TYPE: independent
PROC_TYPE: independent
GROUP: ENGINEERING.SIGNAL_PROCESSING
*)
(*@KEY@:DESCRIPTION*)
version 1.1	18. jan. 2011
programmer 	hugo
tested by	tobias

Scale_B is used to translate and scale a byte input x to a real output.

(*@KEY@:END_DESCRIPTION*)
FUNCTION SCALE_B:REAL

(*Group:Default*)

VAR_INPUT
	X :	BYTE;
	I_LO :	BYTE;
	I_HI :	BYTE;
	O_LO :	REAL;
	O_HI :	REAL;
END_VAR

(*@KEY@: WORKSHEET
NAME: SCALE_B
IEC_LANGUAGE: ST
*)
IF I_HI = I_LO THEN
	SCALE_B := O_LO;
ELSE
	SCALE_B := (O_HI - O_LO) / USINT_TO_REAL(BYTE_TO_USINT(I_HI) - BYTE_TO_USINT(I_LO)) * _BYTE_TO_REAL(LIMIT(I_LO,X,I_HI));
END_IF;

(* revision history
hm	18. may. 2008		rev 1.0
	original version

hm	18. jan 2011		rev 1.1
	avoid division by 0

*)
(*@KEY@: END_WORKSHEET *)
END_FUNCTION

(* ---- SCALE_B2.ST ---- *)
(*@PROPERTIES_EX@
TYPE: POU
LOCALE: 0
IEC_LANGUAGE: ST
PLC_TYPE: independent
PROC_TYPE: independent
GROUP: ENGINEERING.SIGNAL_PROCESSING
*)
(*@KEY@:DESCRIPTION*)
version 1.4	3. nov. 2008
programmer 	hugo
tested by	oscat

this functiob block can scale up to two inputs.
inputs have their min value at 0 and their max value at 255 while the min and max value can be either positive or negative.
inputs ramp between min and max values for the respective inputs to be between (0..255).
the summed output is then scaled by an scale input K and a offset O can be added to the output.
min and max input configurations can be edited in the cfc editor by double clicking the symbol body.
(*@KEY@:END_DESCRIPTION*)
FUNCTION SCALE_B2:REAL

(*Group:Default*)

VAR_INPUT
	IN1 :	BYTE;
	IN2 :	BYTE;
	K :	REAL;(*Standard = 1*)
	O :	REAL;(*Standard = 0*)
	IN1_MIN :	REAL;(*Standard = 0*)
	IN1_MAX :	REAL;(*Standard = 1000*)
	IN2_MIN :	REAL;(*Standard = 0*)
	IN2_MAX :	REAL;(*Standard = 1000*)
END_VAR

(*@KEY@: WORKSHEET
NAME: SCALE_B2
IEC_LANGUAGE: ST
*)
SCALE_B2 := 	(((in1_max - in1_min)* _BYTE_TO_REAL(in1) + (in2_max - in2_min)* _BYTE_TO_REAL(in2)) * 0.003921569 + in1_min + in2_min) * K + O;

(* code bofore rev 1.2
scale_B2 := 	((in1_max - in1_min)* in1 / 255 + in1_min +
				(in2_max - in2_min)* in2 / 255 + in2_min)
				* K + O;
*)

(* revision History
hm 19.1.2007		rev 1.1
	changed outputs to real to avoid overflow of integer
	added offset for better cascading of scale functions
	changed from FB to function

hm	6. jan 2008		rev 1.2
	improved performance

hm	26. oct. 2008	rev 1.3
	code optimization

hm	3. nov. 2008	rev 1.4
	used wrong factor in formula

*)
(*@KEY@: END_WORKSHEET *)
END_FUNCTION

(* ---- SCALE_B4.ST ---- *)
(*@PROPERTIES_EX@
TYPE: POU
LOCALE: 0
IEC_LANGUAGE: ST
PLC_TYPE: independent
PROC_TYPE: independent
GROUP: ENGINEERING.SIGNAL_PROCESSING
*)
(*@KEY@:DESCRIPTION*)
version 1.4	3. nov. 2008
programmer 	hugo
tested by	tobias

	this functiob block can scale up to 4 inputs.
	the inputs have their min value at 0 and their max value at 255 while the min and max value can be either positive or negative.
	the inputs ramp between min and max values for the respective inputs to be between (0..255).
	the summed output is then scaled by an scale input K and a offset O can be added to the output.
	the min and max input configurations can be edited in the cfc editor by double clicking the symbol body.
(*@KEY@:END_DESCRIPTION*)
FUNCTION SCALE_B4:REAL

(*Group:Default*)

VAR_INPUT
	IN1 :	BYTE;
	IN2 :	BYTE;
	IN3 :	BYTE;
	IN4 :	BYTE;
	K :	REAL;(*Standard = 1*)
	O :	REAL;(*Standard = 0*)
	IN1_MIN :	REAL;(*Standard = 0*)
	IN1_MAX :	REAL;(*Standard = 1000*)
	IN2_MIN :	REAL;(*Standard = 0*)
	IN2_MAX :	REAL;(*Standard = 1000*)
	IN3_MIN :	REAL;(*Standard = 0*)
	IN3_MAX :	REAL;(*Standard = 1000*)
	IN4_MIN :	REAL;(*Standard = 0*)
	IN4_MAX :	REAL;(*Standard = 1000*)
END_VAR

(*@KEY@: WORKSHEET
NAME: SCALE_B4
IEC_LANGUAGE: ST
*)
SCALE_B4 := 	(((in1_max - in1_min)* _BYTE_TO_REAL(in1) + (in2_max - in2_min)* _BYTE_TO_REAL(in2) + (in3_max - in3_min)* _BYTE_TO_REAL(in3) + (in4_max - in4_min)* _BYTE_TO_REAL(in4))* 0.003921569 + in1_min + in2_min + in3_min + in4_min) * K + O;

(* revision History
hm 19.1.2007		rev 1.1
	changed outputs to real to avoid overflow of integer
	added offset for better cascading of scale functions
	changed from fb to function

hm	6. jan 2008		rev 1.2
	improved performance

hm	26. oct. 2008	rev 1.3
	optimized code

hm	3. nov. 2008	rev 1.4
	used wrong factor in formula

*)
(*@KEY@: END_WORKSHEET *)
END_FUNCTION

(* ---- SCALE_B8.ST ---- *)
(*@PROPERTIES_EX@
TYPE: POU
LOCALE: 0
IEC_LANGUAGE: ST
PLC_TYPE: independent
PROC_TYPE: independent
GROUP: ENGINEERING.SIGNAL_PROCESSING
*)
(*@KEY@:DESCRIPTION*)
version 1.4	3. nov. 2008
programmer 	hugo
tested by	oscat

this functiob block can scale up to 8 inputs.
the inputs have their min value at 0 and their max value at 255 while the min and max value can be either positive or negative.
the inputs ramp between min and max values for the respective inputs to be between (0..255).
the summed output is then scaled by an scale input K and a offset O can be added to the output.
the min and max input configurations can be edited in the cfc editor by double clicking the symbol body.
(*@KEY@:END_DESCRIPTION*)
FUNCTION SCALE_B8:REAL

(*Group:Default*)

VAR_INPUT
	IN1 :	BYTE;
	IN2 :	BYTE;
	IN3 :	BYTE;
	IN4 :	BYTE;
	IN5 :	BYTE;
	IN6 :	BYTE;
	IN7 :	BYTE;
	IN8 :	BYTE;
	K :	REAL;
	O :	REAL;
	IN1_MIN :	REAL;(*Standard = 0*)
	IN1_MAX :	REAL;(*Standard = 1000*)
	IN2_MIN :	REAL;(*Standard = 0*)
	IN2_MAX :	REAL;(*Standard = 1000*)
	IN3_MIN :	REAL;(*Standard = 0*)
	IN3_MAX :	REAL;(*Standard = 1000*)
	IN4_MIN :	REAL;(*Standard = 0*)
	IN4_MAX :	REAL;(*Standard = 1000*)
	IN5_MIN :	REAL;(*Standard = 0*)
	IN5_MAX :	REAL;(*Standard = 1000*)
	IN6_MIN :	REAL;(*Standard = 0*)
	IN6_MAX :	REAL;(*Standard = 1000*)
	IN7_MIN :	REAL;(*Standard = 0*)
	IN7_MAX :	REAL;(*Standard = 1000*)
	IN8_MIN :	REAL;(*Standard = 0*)
	IN8_MAX :	REAL;(*Standard = 1000*)
END_VAR

(*@KEY@: WORKSHEET
NAME: SCALE_B8
IEC_LANGUAGE: ST
*)
SCALE_B8 := 	(((in1_max - in1_min)* _BYTE_TO_REAL(in1) + (in2_max - in2_min)* _BYTE_TO_REAL(in2) + (in3_max - in3_min)* _BYTE_TO_REAL(in3) + (in4_max - in4_min)* _BYTE_TO_REAL(in4) +
				(in5_max - in5_min)* _BYTE_TO_REAL(in5) + (in6_max - in6_min)* _BYTE_TO_REAL(in6) + (in7_max - in7_min)* _BYTE_TO_REAL(in7) + (in8_max - in8_min)* _BYTE_TO_REAL(in8)) * 0.003921569
				 + in1_min + in2_min + in3_min + in4_min + in5_min + in6_min + in7_min + in8_min) * K + O;

(* revision History
hm	19. jan.2007	rev 1.1
	changed outputs to real to avoid overflow of integer
	added offset for better cascading of scale functions

hm	6. jan. 2008	rev 1.2
	improved performance

hm	26. oct. 2008	rev 1.3
	code optimization

hm	3. nov. 2008	rev 1.4
	used wrong factor in formula

*)
(*@KEY@: END_WORKSHEET *)
END_FUNCTION

(* ---- SCALE_D.ST ---- *)
(*@PROPERTIES_EX@
TYPE: POU
LOCALE: 0
IEC_LANGUAGE: ST
PLC_TYPE: independent
PROC_TYPE: independent
GROUP: ENGINEERING.SIGNAL_PROCESSING
*)
(*@KEY@:DESCRIPTION*)
version 1.2	11. jan. 2011
programmer 	hugo
tested by	oscat

Scale_D is used to translate and scale a DWORD input x to a real output.
the input is limited to I_LO <= X <= I_HI.

(*@KEY@:END_DESCRIPTION*)
FUNCTION SCALE_D:REAL

(*Group:Default*)

VAR_INPUT
	X :	DWORD;
	I_LO :	DWORD;
	I_HI :	DWORD;
	O_LO :	REAL;
	O_HI :	REAL;
END_VAR

(*@KEY@: WORKSHEET
NAME: SCALE_D
IEC_LANGUAGE: ST
*)
IF I_HI = I_LO THEN
	SCALE_D := O_LO;
ELSE
	SCALE_D := (O_HI - O_LO) / UDINT_TO_REAL(DWORD_TO_UDINT(I_HI) - DWORD_TO_UDINT(I_LO)) * UDINT_TO_REAL(LIMIT(DWORD_TO_UDINT(I_LO),DWORD_TO_UDINT(X),DWORD_TO_UDINT(I_HI)) - DWORD_TO_UDINT(I_LO)) + O_LO;
END_IF;

(* revision history
hm	18. may. 2008	rev 1.0
	original version

hm	13. nov. 2008	rev 1.1
	corrected formula for negative gradient

hm	11. jan 2011	rev 1.2
	avoid division by 0
*)
(*@KEY@: END_WORKSHEET *)
END_FUNCTION

(* ---- SCALE_R.ST ---- *)
(*@PROPERTIES_EX@
TYPE: POU
LOCALE: 0
IEC_LANGUAGE: ST
PLC_TYPE: independent
PROC_TYPE: independent
GROUP: ENGINEERING.SIGNAL_PROCESSING
*)
(*@KEY@:DESCRIPTION*)
version 1.2	11. jan. 2011
programmer 	hugo
tested by	oscat

Scale_R is used to translate and scale a REAL input x to a real output.
the input is limited to I_LO <= X <= I_HI.

(*@KEY@:END_DESCRIPTION*)
FUNCTION SCALE_R:REAL

(*Group:Default*)

VAR_INPUT
	X :	REAL;
	I_LO :	REAL;
	I_HI :	REAL;
	O_LO :	REAL;
	O_HI :	REAL;
END_VAR

(*@KEY@: WORKSHEET
NAME: SCALE_R
IEC_LANGUAGE: ST
*)
IF I_LO = I_HI THEN
	SCALE_R := O_LO;
ELSE
	SCALE_R := (O_HI - O_LO) / (I_HI - I_LO) * (LIMIT(I_LO, X, I_HI) - I_LO) + O_LO;
END_IF;

(* revision history
hm	18. may. 2008	rev 1.0
	original version

hm	13. nov. 2008	rev 1.1
	corrected formula for negative gradient

hm	11. jan 2011	rev 1.2
	avoid division by 0

*)
(*@KEY@: END_WORKSHEET *)
END_FUNCTION

(* ---- SCALE_X2.ST ---- *)
(*@PROPERTIES_EX@
TYPE: POU
LOCALE: 0
IEC_LANGUAGE: ST
PLC_TYPE: independent
PROC_TYPE: independent
GROUP: ENGINEERING.SIGNAL_PROCESSING
*)
(*@KEY@:DESCRIPTION*)
version 1.0	19 jan 2007
programmer 	hugo
tested by		tobias

this functiob block can scale up to two inputs.
the input can select between two values with true or false.
the summed output is then scaled by an scale input K and a offset O can be added to the output.
the min and max input configurations can be edited in the cfc editor by double clicking the symbol body.
(*@KEY@:END_DESCRIPTION*)
FUNCTION SCALE_X2:REAL

(*Group:Default*)

VAR_INPUT
	IN1 :	BOOL;
	IN2 :	BOOL;
	K :	REAL;
	O :	REAL;
	IN1_MIN :	REAL;(*Standard = 0*)
	IN1_MAX :	REAL;(*Standard = 1000*)
	IN2_MIN :	REAL;(*Standard = 0*)
	IN2_MAX :	REAL;(*Standard = 1000*)
END_VAR

(*@KEY@: WORKSHEET
NAME: SCALE_X2
IEC_LANGUAGE: ST
*)
SCALE_X2 := (SEL(IN1,IN1_MIN, IN1_MAX)+ SEL(IN2,IN2_MIN, IN2_MAX))* k + o;

(* revision history
hm	19. jan, 2007	rev 1.0
	original version

hm	26. oct. 2008	rev 1.1
	code optimized

*)
(*@KEY@: END_WORKSHEET *)
END_FUNCTION

(* ---- SCALE_X4.ST ---- *)
(*@PROPERTIES_EX@
TYPE: POU
LOCALE: 0
IEC_LANGUAGE: ST
PLC_TYPE: independent
PROC_TYPE: independent
GROUP: ENGINEERING.SIGNAL_PROCESSING
*)
(*@KEY@:DESCRIPTION*)
version 1.0	19 jan 2007
programmer 	hugo
tested by	tobias

this function can scale up to 4 inputs.
the input can select between two values with true or false.
the summed output is then scaled by an scale input K and a offset O can be added to the output.
the min and max input configurations can be edited in the cfc editor by double clicking the symbol body.
(*@KEY@:END_DESCRIPTION*)
FUNCTION SCALE_X4:REAL

(*Group:Default*)

VAR_INPUT
	IN1 :	BOOL;
	IN2 :	BOOL;
	IN3 :	BOOL;
	IN4 :	BOOL;
	K :	REAL;
	O :	REAL;
	IN1_MIN :	REAL;
	IN1_MAX :	REAL;
	IN2_MIN :	REAL;
	IN2_MAX :	REAL;
	IN3_MIN :	REAL;
	IN3_MAX :	REAL;
	IN4_MIN :	REAL;
	IN4_MAX :	REAL;
END_VAR

(*@KEY@: WORKSHEET
NAME: SCALE_X4
IEC_LANGUAGE: ST
*)
IF NOT in1 THEN scale_X4 := in1_min; ELSE scale_X4 := in1_max; END_IF;
IF NOT in2 THEN scale_x4 := scale_x4 + in2_min; ELSE scale_x4 := scale_x4 + in2_max; END_IF;
IF NOT in3 THEN scale_x4 := scale_x4 + in3_min; ELSE scale_x4 := scale_x4 + in3_max; END_IF;
IF NOT in4 THEN scale_x4 := scale_x4 + in4_min; ELSE scale_x4 := scale_x4 + in4_max; END_IF;
scale_X4 := scale_X4 * k + O;
(*@KEY@: END_WORKSHEET *)
END_FUNCTION

(* ---- SCALE_X8.ST ---- *)
(*@PROPERTIES_EX@
TYPE: POU
LOCALE: 0
IEC_LANGUAGE: ST
PLC_TYPE: independent
PROC_TYPE: independent
GROUP: ENGINEERING.SIGNAL_PROCESSING
*)
(*@KEY@:DESCRIPTION*)
version 1.2	24. jan. 2009
programmer 	hugo
tested by	oscat

this function can scale up to 4 inputs.
the input can select between two values with true or false.
the summed output is then scaled by an scale input K and a offset O can be added to the output.
the min and max input configurations can be edited in the cfc editor by double clicking the symbol body.
(*@KEY@:END_DESCRIPTION*)
FUNCTION SCALE_X8:REAL

(*Group:Default*)

VAR_INPUT
	IN1 :	BOOL;
	IN2 :	BOOL;
	IN3 :	BOOL;
	IN4 :	BOOL;
	IN5 :	BOOL;
	IN6 :	BOOL;
	IN7 :	BOOL;
	IN8 :	BOOL;
	K :	REAL;
	O :	REAL;
	IN1_MIN :	REAL;
	IN1_MAX :	REAL;
	IN2_MIN :	REAL;
	IN2_MAX :	REAL;
	IN3_MIN :	REAL;
	IN3_MAX :	REAL;
	IN4_MIN :	REAL;
	IN4_MAX :	REAL;
	IN5_MIN :	REAL;
	IN5_MAX :	REAL;
	IN6_MIN :	REAL;
	IN6_MAX :	REAL;
	IN7_MIN :	REAL;
	IN7_MAX :	REAL;
	IN8_MIN :	REAL;
	IN8_MAX :	REAL;
END_VAR

(*@KEY@: WORKSHEET
NAME: SCALE_X8
IEC_LANGUAGE: ST
*)
SCALE_X8 := (SEL(IN1,IN1_MIN, IN1_MAX)+ SEL(IN2,IN2_MIN, IN2_MAX)+SEL(IN3,IN3_MIN, IN3_MAX)+ SEL(IN4,IN4_MIN, IN4_MAX)
				+SEL(IN5,IN5_MIN, IN5_MAX)+ SEL(IN6,IN6_MIN, IN6_MAX)+SEL(IN7,IN7_MIN, IN7_MAX)+ SEL(IN8,IN8_MIN, IN8_MAX))*k + o;

(* revision history
hm	19. jan. 2008	rev 1.0
	original version

hm	26. oct. 2008	rev 1.1
	optimized code

hm	24. jan. 2008	rev 1.2
	corrected error in formula
*)
(*@KEY@: END_WORKSHEET *)
END_FUNCTION

(* ---- SECOND.ST ---- *)
(*@PROPERTIES_EX@
TYPE: POU
LOCALE: 0
IEC_LANGUAGE: ST
PLC_TYPE: independent
PROC_TYPE: independent
GROUP: TIME_DATE
*)
(*@KEY@:DESCRIPTION*)
version 1.1	2 oct 2006
programmer 	hugo
tested by	tobias

returns the seconds and milliseconds as real of TOD
(*@KEY@:END_DESCRIPTION*)
FUNCTION SECOND:REAL

(*Group:Default*)

VAR_INPUT
	ITOD :	UDINT;
END_VAR

(*@KEY@: WORKSHEET
NAME: SECOND
IEC_LANGUAGE: ST
*)
(*
second := UDINT_TO_REAL(itod - itod/UDINT#60000 * UDINT#60000) / 1000.0;
*)

second := UDINT_TO_REAL(itod MOD UDINT#60000) / REAL#1000.00;

(* change history

2.10.2006 changes name of input to itod

*)
(*@KEY@: END_WORKSHEET *)
END_FUNCTION

(* ---- SECOND_OF_DT.ST ---- *)
(*@PROPERTIES_EX@
TYPE: POU
LOCALE: 0
IEC_LANGUAGE: ST
PLC_TYPE: independent
PROC_TYPE: independent
GROUP: TIME_DATE
*)
(*@KEY@:DESCRIPTION*)
version 1.0	6. jun. 2008
programmer 	oscat
tested BY	oscat

SECOND_OF_DT returns the current second (second of minute) of a DT variable
(*@KEY@:END_DESCRIPTION*)
FUNCTION SECOND_OF_DT:INT

(*Group:Default*)

VAR_INPUT
	XDT :	UDINT;
END_VAR

(*@KEY@: WORKSHEET
NAME: SECOND_OF_DT
IEC_LANGUAGE: ST
*)
SECOND_OF_DT := UDINT_TO_INT(XDT MOD UDINT#60);

(* revision history
hm		6.9.2008	rev 1.0
	original version

*)
(*@KEY@: END_WORKSHEET *)
END_FUNCTION

(* ---- SECOND_TO_TIME.ST ---- *)
(*@PROPERTIES_EX@
TYPE: POU
LOCALE: 0
IEC_LANGUAGE: ST
PLC_TYPE: independent
PROC_TYPE: independent
GROUP: TIME_DATE
*)
(*@KEY@:DESCRIPTION*)
version 1.2	24. feb. 2009
programmer 	hugo
tested by	tobias

converts an amount of seconds in real to time
(*@KEY@:END_DESCRIPTION*)
FUNCTION SECOND_TO_TIME:TIME

(*Group:Default*)

VAR_INPUT
	IN :	REAL;
END_VAR

(*@KEY@: WORKSHEET
NAME: SECOND_TO_TIME
IEC_LANGUAGE: ST
*)
second_to_time := UDINT_TO_TIME(_REAL_TO_UDINT(IN * 1000.0));

(* revision history
hm		4. aug 2006	rev 1.0
	original version

hm		14. mar 2008	rev 1.1
	rounded the input after the last digit
*)
(*@KEY@: END_WORKSHEET *)
END_FUNCTION

(* ---- SENSOR_INT.ST ---- *)
(*@PROPERTIES_EX@
TYPE: POU
LOCALE: 0
IEC_LANGUAGE: ST
PLC_TYPE: independent
PROC_TYPE: independent
GROUP: ENGINEERING.SENSOR
*)
(*@KEY@:DESCRIPTION*)
version 1.3	11. mar. 2009
programmer 	hugo
tested by	tobias

this function calculates the real resistance of a sensor RX given a parasitic resistor in parallel to the sensor and an additional serial resistor.
for example a parasitic parallel resistor for a PT100 can be ignored but a series resistor is the cable to the sensor.
for a humidity sensor, the parallel resistor is more dramatic and needs to be considered.
the function allows to consider a parallel and serial resistor at the same time.
with this function and known parasitic serial and parallel resistors the true resistance of the sensor can be calculated.

(*@KEY@:END_DESCRIPTION*)
FUNCTION SENSOR_INT:REAL

(*Group:Default*)

VAR_INPUT
	VOLTAGE :	REAL;
	CURRENT :	REAL;
	RP :	REAL;
	RS :	REAL;
END_VAR

VAR
	RG :	REAL;
END_VAR

(*@KEY@: WORKSHEET
NAME: SENSOR_INT
IEC_LANGUAGE: ST
*)
IF current <> 0.0 THEN
	RG := voltage / current;
	SENSOR_INT := RP * ( RG - RS) / ( RP + RS - RG);
END_IF;

(* revisaion history

hm 20.1.2007		rev 1.1
	deleted input R0 which was not needed.

hm	2. dec 2007	rev 1.2
	corrected an error in formula and improoved speed

hm	11. mar. 2009	rev 1.3
	changed real constants to use dot syntax

*)
(*@KEY@: END_WORKSHEET *)
END_FUNCTION

(* ---- SET_DATE.ST ---- *)
(*@PROPERTIES_EX@
TYPE: POU
LOCALE: 0
IEC_LANGUAGE: ST
PLC_TYPE: independent
PROC_TYPE: independent
GROUP: TIME_DATE
*)
(*@KEY@:DESCRIPTION*)
version 2.3	29. dec. 2011
programmer 	hugo
tested by	tobias

creates a date output from year, month and day of month

(*@KEY@:END_DESCRIPTION*)
FUNCTION SET_DATE:UDINT

(*Group:default*)

VAR_INPUT
	YEAR :	INT;
	MONTH :	INT;
	DAY :	INT;
END_VAR

VAR
	count :	INT;
END_VAR

(*@KEY@: WORKSHEET
NAME: SET_DATE
IEC_LANGUAGE: ST
*)
IF month > 2 THEN
	count := (month - 1) * 30;
	IF month > 7 THEN
		count := count + DWORD_TO_INT(SHR_DWORD(DINT_TO_DWORD(INT_TO_DINT(month) - INT_TO_DINT(3)),1));
	ELSE
		count := count + DWORD_TO_INT(SHR_DWORD(DINT_TO_DWORD(INT_TO_DINT(month) - INT_TO_DINT(4)),1));
	END_IF;
	(* chech for leap year and add one day if true *)
	IF SHL_WORD(INT_TO_WORD(year),14) = WORD#0 THEN
		count := count + 1;
	END_IF;
ELSE
	count := (month - 1) * 31;
END_IF;
SET_DATE := (_INT_TO_UDINT(count + day - 1) + DWORD_TO_UDINT(SHR(UDINT_TO_DWORD(_INT_TO_UDINT(year) * UDINT#1461 - UDINT#2878169), 2))) * UDINT#86400;

(* revision history
hm	4. aug. 2006	rev 1.0
	original version

hm	19 sep. 2007	rev 1.1
	use function leap_year to calculate leap year, more exceptions are handled

hm	1. okt	2007	rev 1.2
	added compatibility to step7

hm	16.dec 2007		rev 1.3
	changed code to improove performance

hm	3. jan. 2008	rev 1.4
	further improvements in performance

hm	16. mar. 2008	rev 1.5
	added type conversions to avoid warnings under codesys 3.0

hm	7. apr. 2008	rev 1.6
	deleted unused step7 code

hm	14. oct. 2008	rev 1.7
	optimized code for better performance

hm	25. oct. 2008	rev 2.0
	new code using setup constants

hm	16. nov. 2008	rev 2.1
	added typecasts to avoid warnings

hm	22. jan. 2011	rev 2.2
	improved performance

hm	29. dec. 2011	rev 2.3
	improved performance
*)

(*@KEY@: END_WORKSHEET *)
END_FUNCTION

(* ---- SET_DT.ST ---- *)
(*@PROPERTIES_EX@
TYPE: POU
LOCALE: 0
IEC_LANGUAGE: ST
PLC_TYPE: independent
PROC_TYPE: independent
GROUP: TIME_DATE
*)
(*@KEY@:DESCRIPTION*)
version 1.5	16 mar 2008
programmer 	hugo
tested by	tobias

creates a date output from year, month and day of month
year must be in the form of 4 digits ie 2006 or 1977.
(*@KEY@:END_DESCRIPTION*)
FUNCTION SET_DT:UDINT

(*Group:Default*)

VAR_INPUT
	YEAR :	INT;
	MONTH :	INT;
	DAY :	INT;
	HOUR :	INT;
	MINUTE :	INT;
	SECOND :	INT;
END_VAR

(*@KEY@: WORKSHEET
NAME: SET_DT
IEC_LANGUAGE: ST
*)
SET_DT := SET_DATE(YEAR, MONTH, DAY) + _INT_TO_UDINT(SECOND) + _INT_TO_UDINT(MINUTE) * UDINT#60 + _INT_TO_UDINT(HOUR) * UDINT#3600;

(* revision history
hm	4. aug. 2006		rev 1.0
	original version

hm		19 sep. 2007	rev 1.1
	use function leap_year to calculate leap year, more exceptions are handled

hm		1. okt 2007		rev 1.2
	added step7 compatibility
	call function set_date

hm		8. oct 2007		rev 1.3
	deleted unused variables count and leap

hm		1. 11 2007		rev 1.4
	converted hour type integer to dword in calculation to avoid overrun on möller ecp4

hm		16. mar 2008	rev 1.5
	added type conversions to avoid warnings under codesys 3.0
*)

(*@KEY@: END_WORKSHEET *)
END_FUNCTION

(* ---- SET_TOD.ST ---- *)
(*@PROPERTIES_EX@
TYPE: POU
LOCALE: 0
IEC_LANGUAGE: ST
PLC_TYPE: independent
PROC_TYPE: independent
GROUP: TIME_DATE
*)
(*@KEY@:DESCRIPTION*)
version 1.5	16. mar 2008
programmer 	hugo
tested by	tobias

creates tod from hour minute and second
(*@KEY@:END_DESCRIPTION*)
FUNCTION SET_TOD:UDINT

(*Group:Default*)

VAR_INPUT
	HOUR :	INT;
	MINUTE :	INT;
	SECOND :	REAL;
END_VAR

(*@KEY@: WORKSHEET
NAME: SET_TOD
IEC_LANGUAGE: ST
*)
set_Tod := _REAL_TO_UDINT(second * 1000.0) + _INT_TO_UDINT(minute) * UDINT#60000 + _INT_TO_UDINT(hour) * UDINT#3600000;

(* revision history

hm		4.aug.2006		rev 1.0
	original version

hm		11. sep 2007	rev 1.1
	changed coding to avoid a compiler warning under twincat.

hm		1. nov 2007	rev 1.2
	changed coding to avoid possible overrun situation on möller ecp4

hm		2. Nov	2007	rev 1.3
	changed dword to DINT in calcualtion to avoid warnings with some compilers

hm		14. mar 2008	rev 1.4
	changed code to avoid rounding problem at last digit of millisecond

hm		16. mar. 2008	rev 1.5
	added type conversions to avoid warning under codesys 3.0
*)
(*@KEY@: END_WORKSHEET *)
END_FUNCTION

(* ---- SGN.ST ---- *)
(*@PROPERTIES_EX@
TYPE: POU
LOCALE: 0
IEC_LANGUAGE: ST
PLC_TYPE: independent
PROC_TYPE: independent
GROUP: MATHEMATICAL.MATHE
*)
(*@KEY@:DESCRIPTION*)
version 1.1	11 nov 2007
programmer 	hugo
tested by	tobias

sgn returns 0 when X = 0 , -1 when X < 1 and +1 when X > 1
(*@KEY@:END_DESCRIPTION*)
FUNCTION SGN:INT

(*Group:Default*)

VAR_INPUT
	X :	REAL;
END_VAR

(*@KEY@: WORKSHEET
NAME: SGN
IEC_LANGUAGE: ST
*)
IF X > 0.0 THEN
	sgn := 1;
ELSIF X < 0.0 THEN
	sgn := -1;
ELSE
	sgn := 0;
END_IF;

(* revision histroy
hm	16. oct 2007	rev 1.0
	original version

hm	11. nov 2007	rev 1.1
	changed type of function from real to int
*)
(*@KEY@: END_WORKSHEET *)
END_FUNCTION

(* ---- SHL1.ST ---- *)
(*@PROPERTIES_EX@
TYPE: POU
LOCALE: 0
IEC_LANGUAGE: ST
PLC_TYPE: independent
PROC_TYPE: independent
GROUP: LOGIC.GATE_LOGIC
*)
(*@KEY@:DESCRIPTION*)
version 1.1	27 dec 2007
programmer 	hugo
tested by	tobias

SHL1 shifts N bits to the left filling the new bits with 1
(*@KEY@:END_DESCRIPTION*)
FUNCTION SHL1:DWORD

(*Group:Default*)

VAR_INPUT
	IN :	DWORD;
	N :	INT;
END_VAR

(*@KEY@: WORKSHEET
NAME: SHL1
IEC_LANGUAGE: ST
*)
SHL1 := SHR(DWORD#16#FF_FF_FF_FF,32-N) OR SHL(IN,N);

(* revision history
hm	14.9.2007		rev 1.0
	original version

hm	27. dec 2007	rev 1.1
	changed code for better performance

*)
(*@KEY@: END_WORKSHEET *)
END_FUNCTION

(* ---- SHR1.ST ---- *)
(*@PROPERTIES_EX@
TYPE: POU
LOCALE: 0
IEC_LANGUAGE: ST
PLC_TYPE: independent
PROC_TYPE: independent
GROUP: LOGIC.GATE_LOGIC
*)
(*@KEY@:DESCRIPTION*)
version 1.1	27 dec 2007
programmer 	hugo
tested by	tobias

SHR1 shifts N bits to the right filling the new bits with 1
(*@KEY@:END_DESCRIPTION*)
FUNCTION SHR1:DWORD

(*Group:Default*)

VAR_INPUT
	IN :	DWORD;
	N :	INT;
END_VAR

(*@KEY@: WORKSHEET
NAME: SHR1
IEC_LANGUAGE: ST
*)
SHR1 := SHL(DWORD#16#FF_FF_FF_FF,32-N) OR SHR(IN,N);

(* revision history
hm	14.9.2007		rev 1.0
	original version

hm	27. dec 2007	rev 1.1
	changed code for better performance

*)
(*@KEY@: END_WORKSHEET *)
END_FUNCTION

(* ---- SIGMOID.ST ---- *)
(*@PROPERTIES_EX@
TYPE: POU
LOCALE: 0
IEC_LANGUAGE: ST
PLC_TYPE: independent
PROC_TYPE: independent
GROUP: MATHEMATICAL.MATHE
*)
(*@KEY@:DESCRIPTION*)
version 1.2	10. mar. 2009
programmer 	hugo
tested by	tobias

this function calculates the sigmoid function

(*@KEY@:END_DESCRIPTION*)
FUNCTION SIGMOID:REAL

(*Group:Default*)

VAR_INPUT
	X :	REAL;
END_VAR

(*@KEY@: WORKSHEET
NAME: SIGMOID
IEC_LANGUAGE: ST
*)
IF X > 20.0 THEN
	SIGMOID := 1.0;
ELSIF x < -85.0 THEN
	SIGMOID := 0.0;
ELSE
	SIGMOID := 1.0 / (1.0 + EXP(-X));
END_IF;

(* revision history
hm	10.12.2007		rev 1.0
	original version

hm	11. mar. 2008		rev 1.1
	extended range of valid inputs to +inv / -inv

hm 10. mar. 2009		rev 1.2
	real constants updated to new systax using dot

*)
(*@KEY@: END_WORKSHEET *)
END_FUNCTION

(* ---- SIGN_I.ST ---- *)
(*@PROPERTIES_EX@
TYPE: POU
LOCALE: 0
IEC_LANGUAGE: ST
PLC_TYPE: independent
PROC_TYPE: independent
GROUP: MATHEMATICAL.MATHE
*)
(*@KEY@:DESCRIPTION*)
version 1.3	27. oct. 2008
programmer 	hugo
tested by	tobias

this function return true if the integer input is negative
(*@KEY@:END_DESCRIPTION*)
FUNCTION SIGN_I:BOOL

(*Group:Default*)

VAR_INPUT
	IN :	DINT;
END_VAR

(*@KEY@: WORKSHEET
NAME: SIGN_I
IEC_LANGUAGE: ST
*)
sign_I := BIT_OF_DWORD(DINT_TO_DWORD(in),31);

(* revision history
hm 3.3.2007	rev 1.1
	changed method of function for better compatibility to other systems

hm	1.12.2007	rev 1.2
	changed code to improve performance

hm	27. oct. 2008	rev 1.3
	changed type of input to dint
*)
(*@KEY@: END_WORKSHEET *)
END_FUNCTION

(* ---- SIGN_R.ST ---- *)
(*@PROPERTIES_EX@
TYPE: POU
LOCALE: 0
IEC_LANGUAGE: ST
PLC_TYPE: independent
PROC_TYPE: independent
GROUP: MATHEMATICAL.MATHE
*)
(*@KEY@:DESCRIPTION*)
version 1.4	10. mar. 2009
programmer 	hugo
tested by	tobias

this function return true if the real input is negative
(*@KEY@:END_DESCRIPTION*)
FUNCTION SIGN_R:BOOL

(*Group:Default*)

VAR_INPUT
	IN :	REAL;
END_VAR

(*@KEY@: WORKSHEET
NAME: SIGN_R
IEC_LANGUAGE: ST
*)
SIGN_R := in < 0.0;

(* revision history
hm 19.1.2007	rev 1.1
	changed method of function for better compatibility to other systems

hm	1.12.2007	rev 1.2
	changed code to improve performance

hm	14. jun. 2008	rev 1.3
	improved performace

hm 10. mar. 2009	rev 1.4
	real constants updated to new systax using dot

*)
(*@KEY@: END_WORKSHEET *)
END_FUNCTION

(* ---- SINC.ST ---- *)
(*@PROPERTIES_EX@
TYPE: POU
LOCALE: 0
IEC_LANGUAGE: ST
PLC_TYPE: independent
PROC_TYPE: independent
GROUP: MATHEMATICAL.MATHE
*)
(*@KEY@:DESCRIPTION*)
version 1.2	10. mar. 2009
programmer 	hugo
tested by	tobias

this function calculates the sinc function.
(*@KEY@:END_DESCRIPTION*)
FUNCTION SINC:REAL

(*Group:Default*)

VAR_INPUT
	X :	REAL;
END_VAR

(*@KEY@: WORKSHEET
NAME: SINC
IEC_LANGUAGE: ST
*)
IF X = 0.0 THEN
	SINC := 1.0;
ELSE
	SINC := SIN(x) / x;
END_IF;

(* revision histroy
hm	11. mar. 2008	rev 1.0
	original version

hm	1.12.2007	rev 1.1
	changed code to improove performance

hm 10. mar. 2009	rev 1.2
	real constants updated to new systax using dot

*)
(*@KEY@: END_WORKSHEET *)
END_FUNCTION

(* ---- SINH.ST ---- *)
(*@PROPERTIES_EX@
TYPE: POU
LOCALE: 0
IEC_LANGUAGE: ST
PLC_TYPE: independent
PROC_TYPE: independent
GROUP: MATHEMATICAL.MATHE
*)
(*@KEY@:DESCRIPTION*)
version 1.3	11. mar 2008
programmer 	hugo
tested by	tobias

this function calculates the sin hyperbolicus
(*@KEY@:END_DESCRIPTION*)
FUNCTION SINH:REAL

(*Group:Default*)

VAR_INPUT
	X :	REAL;
END_VAR

(*@KEY@: WORKSHEET
NAME: SINH
IEC_LANGUAGE: ST
*)
IF ABS(x) < 2.0E-3 THEN
	SINH := X;
ELSE
	SINH := (EXP(x) - EXP(-x)) * 0.5;
END_IF;

(* revision history
hm	12.1.2007	rev 1.0
	original version

hm	1.12.2007	rev 1.1
	changed code to improve performance

hm	5. jan 2008	rev 1.2
	further performance improvement

hm	11. mar 2008	rev 1.3
	improved accuracy around 0

*)
(*@KEY@: END_WORKSHEET *)
END_FUNCTION

(* ---- SPHERE_V.ST ---- *)
(*@PROPERTIES_EX@
TYPE: POU
LOCALE: 0
IEC_LANGUAGE: ST
PLC_TYPE: independent
PROC_TYPE: independent
GROUP: MATHEMATICAL.GEOMETRY
*)
(*@KEY@:DESCRIPTION*)
version 1.2	22. feb 2008
programmer 	hugo
tested by	tobias

sphere_V calculates the Volume of a Sphere
(*@KEY@:END_DESCRIPTION*)
FUNCTION SPHERE_V:REAL

(*Group:Default*)

VAR_INPUT
	RX :	REAL;
END_VAR

(*@KEY@: WORKSHEET
NAME: SPHERE_V
IEC_LANGUAGE: ST
*)
sphere_V := 4.188790205 * Rx * RX * RX;

(* revision histroy
hm	16. oct 2007	rev 1.0
	original version

hm	4. dec 2007		rev 1.1
	changed code for better performance

hm	22. feb 2008		rev 1.2
	changed code for better performance
*)
(*@KEY@: END_WORKSHEET *)
END_FUNCTION

(* ---- SQRTN.ST ---- *)
(*@PROPERTIES_EX@
TYPE: POU
LOCALE: 0
IEC_LANGUAGE: ST
PLC_TYPE: independent
PROC_TYPE: independent
GROUP: MATHEMATICAL.MATHE
*)
(*@KEY@:DESCRIPTION*)
version 1.3	10. mar. 2009
programmer 	hugo
tested by	tobias

this function calculates the nth root function of X according to the formula sqrtn = x^(1/n).

(*@KEY@:END_DESCRIPTION*)
FUNCTION SQRTN:REAL

(*Group:Default*)

VAR_INPUT
	X :	REAL;
	N :	INT;
END_VAR

(*@KEY@: WORKSHEET
NAME: SQRTN
IEC_LANGUAGE: ST
*)
IF N > 0 THEN
	SQRTN := EXP(LN(x) / INT_TO_REAL(n));
ELSE
	SQRTN := 0.0;
END_IF;

(* revision history
hm		12 jan 2007	rev 1.0
	original version

hm		2. dec 2007	rev 1.1
	changed code for better performance

hm		11. mar 2008	rev 1.2
	added result 0 for compatibility reasons

hm 10. mar. 2009	rev 1.3
	added type conversions for compatibility reasons

*)
(*@KEY@: END_WORKSHEET *)
END_FUNCTION

(* ---- STAIR.ST ---- *)
(*@PROPERTIES_EX@
TYPE: POU
LOCALE: 0
IEC_LANGUAGE: ST
PLC_TYPE: independent
PROC_TYPE: independent
GROUP: ENGINEERING.SIGNAL_PROCESSING
*)
(*@KEY@:DESCRIPTION*)
version 1.4	10. mar. 2009
programmer 	oscat
tested by	tobias

the function stair converts an anlog input signal to a staircase like output.
D is the step width for the output signal.
if D = 0 then the output follows the input without a chage.
(*@KEY@:END_DESCRIPTION*)
FUNCTION STAIR:REAL

(*Group:Default*)

VAR_INPUT
	X :	REAL;
	D :	REAL;
END_VAR

(*@KEY@: WORKSHEET
NAME: STAIR
IEC_LANGUAGE: ST
*)
IF D > 0.0 THEN
	STAIR := DINT_TO_REAL(_REAL_TO_DINT(X / D)) * D;
ELSE
	STAIR := X;
END_IF;

(* revision history
hm	28 jan 2007		rev 1.0
	original version

hm	27 dec 2007		rev 1.1
	changed code for better performance

hm	6. jan 2008		rev 1.2
	further performance improvement

hm	26. oct. 2008		rev 1.3
	optimized code

hm	10. mar. 2009	rev 1.4
	real constants updated to new systax using dot

*)
(*@KEY@: END_WORKSHEET *)
END_FUNCTION

(* ---- SUN_MIDDAY.ST ---- *)
(*@PROPERTIES_EX@
TYPE: POU
LOCALE: 0
IEC_LANGUAGE: ST
PLC_TYPE: independent
PROC_TYPE: independent
GROUP: TIME_DATE
*)
(*@KEY@:DESCRIPTION*)
version 1.0	26. jan. 2011
programmer 	hugo
tested by	oscat

this FUNCTION calculates the time when the sun stand exactly south of a given location.
(*@KEY@:END_DESCRIPTION*)
FUNCTION SUN_MIDDAY:UDINT

(*Group:Default*)

VAR_INPUT
	LON :	REAL;
	UTC :	UDINT;
END_VAR

VAR
	T :	REAL;
	OFFSET :	REAL;
END_VAR

(*@KEY@: WORKSHEET
NAME: SUN_MIDDAY
IEC_LANGUAGE: ST
*)
T := INT_TO_REAL(DAY_OF_YEAR(utc));
OFFSET := -0.1752 * SIN(0.033430 * T + 0.5474) - 0.1340 * SIN(0.018234 * T - 0.1939);
SUN_MIDDAY := HOUR_TO_TOD(12.0 - OFFSET - lon * 0.0666666666666);

(* revision history

hm	26. jan. 2011	rev 1.0
	initial release

*)

(*@KEY@: END_WORKSHEET *)
END_FUNCTION

(* ---- SWAP_BYTE.ST ---- *)
(*@PROPERTIES_EX@
TYPE: POU
LOCALE: 0
IEC_LANGUAGE: ST
PLC_TYPE: independent
PROC_TYPE: independent
GROUP: LOGIC.GATE_LOGIC
*)
(*@KEY@:DESCRIPTION*)
version 1.0	4 feb 2008
programmer 	hugo
tested by	tobias

This function swaps the high and low byte of the word in.
(*@KEY@:END_DESCRIPTION*)
FUNCTION SWAP_BYTE:WORD

(*Group:Default*)

VAR_INPUT
	IN :	WORD;
END_VAR

(*@KEY@: WORKSHEET
NAME: SWAP_BYTE
IEC_LANGUAGE: ST
*)
Swap_Byte := ROL_WORD(in,8);

(* revision history
hm		4. feb 2008	rev 1.0
	original version

*)
(*@KEY@: END_WORKSHEET *)
END_FUNCTION

(* ---- SWAP_BYTE2.ST ---- *)
(*@PROPERTIES_EX@
TYPE: POU
LOCALE: 0
IEC_LANGUAGE: ST
PLC_TYPE: independent
PROC_TYPE: independent
GROUP: LOGIC.GATE_LOGIC
*)
(*@KEY@:DESCRIPTION*)
version 1.0	4 feb 2008
programmer 	hugo
tested by	tobias

This function reverses the byte order in the dword.
(*@KEY@:END_DESCRIPTION*)
FUNCTION SWAP_BYTE2:DWORD

(*Group:Default*)

VAR_INPUT
	IN :	DWORD;
END_VAR

(*@KEY@: WORKSHEET
NAME: SWAP_BYTE2
IEC_LANGUAGE: ST
*)
Swap_Byte2 := (ROR_DWORD(in,8) AND DWORD#16#FF00FF00) OR (ROL_DWORD(in,8) AND DWORD#16#00FF00FF);

(* revision history
hm		4. feb 2008	rev 1.0
	original version

*)
(*@KEY@: END_WORKSHEET *)
END_FUNCTION

(* ---- TANC.ST ---- *)
(*@PROPERTIES_EX@
TYPE: POU
LOCALE: 0
IEC_LANGUAGE: ST
PLC_TYPE: independent
PROC_TYPE: independent
GROUP: MATHEMATICAL.MATHE
*)
(*@KEY@:DESCRIPTION*)
version 1.1	10. mar. 2009
programmer 	hugo
tested by	oscat

this function calculates the tanc function.

(*@KEY@:END_DESCRIPTION*)
FUNCTION TANC:REAL

(*Group:Default*)

VAR_INPUT
	X :	REAL;
END_VAR

(*@KEY@: WORKSHEET
NAME: TANC
IEC_LANGUAGE: ST
*)
IF X = 0.0 THEN
	TANC := 1.0;
ELSE
	TANC := TAN(x) / x;
END_IF;

(* revision histroy
hm	23. oct. 2008	rev 1.0
	original version

hm 10. mar. 2009	rev 1.1
	real constants updated to new systax using dot

*)
(*@KEY@: END_WORKSHEET *)
END_FUNCTION

(* ---- TANH.ST ---- *)
(*@PROPERTIES_EX@
TYPE: POU
LOCALE: 0
IEC_LANGUAGE: ST
PLC_TYPE: independent
PROC_TYPE: independent
GROUP: MATHEMATICAL.MATHE
*)
(*@KEY@:DESCRIPTION*)
version 1.3	10. mar. 2009
programmer 	hugo
tested by	tobias

this function calculates the tangens hyperbolicus
(*@KEY@:END_DESCRIPTION*)
FUNCTION TANH:REAL

(*Group:Default*)

VAR_INPUT
	X :	REAL;
END_VAR

(*@KEY@: WORKSHEET
NAME: TANH
IEC_LANGUAGE: ST
*)
IF X > 20.0 THEN
	TANH := 1.0;
ELSIF X < -20.0 THEN
	TANH := -1.0;
ELSE
	TANH := 1.0 - 2.0 / (EXP(2.0 * x) + 1.0);
END_IF;

(* revision hisdtory
hm		12.1.2007		rev 1.0
	original version

hm		1.12.2007		rev 1.1
	changed code to improve performance

hm		10. mar 2008	rev 1.2
	corrected an error in formula
	extended range of valid inputs to +/- INV

hm 10. mar. 2009	rev 1.3
	real constants updated to new systax using dot

*)
(*@KEY@: END_WORKSHEET *)
END_FUNCTION

(* ---- TEMP_NI.ST ---- *)
(*@PROPERTIES_EX@
TYPE: POU
LOCALE: 0
IEC_LANGUAGE: ST
PLC_TYPE: independent
PROC_TYPE: independent
GROUP: ENGINEERING.SENSOR
*)
(*@KEY@:DESCRIPTION*)
version 1.5	10. mar. 2009
programmer 	hugo
tested by	tobias

this function returns the temperature for a nickel sensor in a range from -60..+180 °C *)
(*@KEY@:END_DESCRIPTION*)
FUNCTION TEMP_NI:REAL

(*Group:Default*)

VAR_INPUT
	RES :	REAL;
	R0 :	REAL;
END_VAR

(*@KEY@: WORKSHEET
NAME: TEMP_NI
IEC_LANGUAGE: ST
*)
TEMP_NI := (SQRT(0.30085225 - 2.66E-3 * (R0 - Res)) - 0.5485) * 751.8796992;

(* revision history

hm 24.1.2007		rev 1.1
	deleted unused variable A, B, C

hm 10.9.2007		rev 1.2
	changed accuracy to 0.02 degrees to improove performace

hm 17. 12 2007	rev 1.3
	improovements for better performance and higher accuracy

hm	6. jan 2008	rev 1.4
	further performance improvement

hm	10. mar. 2009	rev 1.5
	removed nested comments

*)

(*@KEY@: END_WORKSHEET *)
END_FUNCTION

(* ---- TEMP_NTC.ST ---- *)
(*@PROPERTIES_EX@
TYPE: POU
LOCALE: 0
IEC_LANGUAGE: ST
PLC_TYPE: independent
PROC_TYPE: independent
GROUP: ENGINEERING.SENSOR
*)
(*@KEY@:DESCRIPTION*)
version 1.1	11. mar. 2009
programmer 	hugo
tested by	tobias

this function returs the temperature for a NTC sensor for a range from 0..85 °C.
RN is the resistance at 25 °C and B is a constant for the given sensor.

(*@KEY@:END_DESCRIPTION*)
FUNCTION TEMP_NTC:REAL

(*Group:Default*)

VAR_INPUT
	RES :	REAL;
	RN :	REAL;
	B :	REAL;
END_VAR

(*@KEY@: WORKSHEET
NAME: TEMP_NTC
IEC_LANGUAGE: ST
*)
IF res > 0.0 THEN
	TEMP_NTC := B * 298.15 / (B + LN(RES / RN) * 298.15) -273.15;
END_IF;

(* revision history

hm 30. dec. 2008	rev 1.0
	original version

hm	11. mar. 2009	rev 1.1
	changed real constants to use dot syntax

*)
(*@KEY@: END_WORKSHEET *)
END_FUNCTION

(* ---- TEMP_PT.ST ---- *)
(*@PROPERTIES_EX@
TYPE: POU
LOCALE: 0
IEC_LANGUAGE: ST
PLC_TYPE: independent
PROC_TYPE: independent
GROUP: ENGINEERING.SENSOR
*)
(*@KEY@:DESCRIPTION*)
version 1.7	11. mar. 2009
programmer 	hugo
tested by		oscat

this function returs the temperature for a platinum sensor for a range from -200..+850 °C

(*@KEY@:END_DESCRIPTION*)
FUNCTION TEMP_PT:REAL

(*Group:Default*)

VAR_INPUT
	RES :	REAL;
	R0 :	REAL;
END_VAR

VAR
	step :	REAL := REAL#50.0;
	X :	REAL;
	Y :	REAL;
	t1 :	REAL;
END_VAR

(*@KEY@: WORKSHEET
NAME: TEMP_PT
IEC_LANGUAGE: ST
*)
X := 3.9083E-3 * R0;
Y := -5.775E-7 * R0;
IF Res >= R0 THEN
	t1 := X * X - 4.0 * Y * (R0 - Res);
	IF t1 < 0.0 THEN
		TEMP_PT := 10000.0;
	ELSE
		TEMP_PT := (-X + SQRT(t1)) / (2.0 * Y);
	END_IF;
ELSE
	(* since the formula cannot be solved this is a successive approximation *)
	TEMP_PT := -100.0;
	WHILE step > 0.01 DO
		(* test if result greater or less *)
		IF RES_PT(TEMP_PT, R0) < res THEN TEMP_PT := TEMP_PT + step; ELSE TEMP_PT := TEMP_PT - step; END_IF;
		step := step * 0.5;
	END_WHILE;
END_IF;

(* revision history

rev 1.1 hm 24.1.2007
	deleted unused variable C

rev 1.2 hm 10.9.2007
	reduced accuracy to 0.02 to shorten execution time

rev 1.3	hm	2. dec 2007
	changed code for better performance

rev	1.4	hm	23. dec 2007
	avoid a negative square root if input values are wrong

rev 1.5 hm	5. jan 2008
	replaced / 2 with * 0.5 for better performance

hm	31. oct. 2008	rev 1.6
	improved performance

hm	11. mar. 2009	rev 1.7
	changed real constants to use dot syntax

*)

(*@KEY@: END_WORKSHEET *)
END_FUNCTION

(* ---- TEMP_SI.ST ---- *)
(*@PROPERTIES_EX@
TYPE: POU
LOCALE: 0
IEC_LANGUAGE: ST
PLC_TYPE: independent
PROC_TYPE: independent
GROUP: ENGINEERING.SENSOR
*)
(*@KEY@:DESCRIPTION*)
version 1.5	10. mar. 2009
programmer 	hugo
tested by	tobias

this function returs the temperature for a silicon sensor for a range from -60..+180 °C
for example KTY10 RS at TS normally 25 °C

(*@KEY@:END_DESCRIPTION*)
FUNCTION TEMP_SI:REAL

(*Group:Default*)

VAR_INPUT
	RES :	REAL;
	RS :	REAL;
	TS :	REAL;
END_VAR

(*@KEY@: WORKSHEET
NAME: TEMP_SI
IEC_LANGUAGE: ST
*)
TEMP_SI := (-7.64E-3 + SQRT(Res/RS* 6.64E-5 - 0.803E-5)) * 30120.48193 + TS;

(* revision history

hm 24.1.2007		rev 1.1
	the function would only work for TS = 25, now it works for other values of ts.

hm 10.9.2007		rev 1.2
	changed the function to use successive approcimation to avoid an error generated by a sqrt from a negative result.
	changed accuracy to 0.02 degrees to shorten execution time

hm 17. 12 2007	rev 1.3
	improovements for better performance

hm	6. jan 2008	rev 1.4
	further performance improvement

hm	10. mar. 2009	rev 1.5
	removed nested comments

*)
(*@KEY@: END_WORKSHEET *)
END_FUNCTION

(* ---- TIMECHECK.ST ---- *)
(*@PROPERTIES_EX@
TYPE: POU
LOCALE: 0
IEC_LANGUAGE: ST
PLC_TYPE: independent
PROC_TYPE: independent
GROUP: TIME_DATE
*)
(*@KEY@:DESCRIPTION*)
version 1.0	19. jul. 2009
programmer 	oscat
tested by	oscat

this function retruns true if the daytime TD is between start and stop and returns true if so.
if you want to generate an event to span over midnight, start timemust be later than the stop time.

(*@KEY@:END_DESCRIPTION*)
FUNCTION TIMECHECK:BOOL

(*Group:Default*)

VAR_INPUT
	TD :	UDINT;
	START :	UDINT;
	STOP :	UDINT;
END_VAR

(*@KEY@: WORKSHEET
NAME: TIMECHECK
IEC_LANGUAGE: ST
*)
IF stop < start THEN
	TIMECHECK := start <= TD OR  TD < stop;
ELSE
	TIMECHECK := start <= TD AND TD < stop;
END_IF;

(* revision history
hm 19. jul. 2009	rev 1.0
	original release

*)
(*@KEY@: END_WORKSHEET *)
END_FUNCTION

(* ---- TO_LOWER.ST ---- *)
(*@PROPERTIES_EX@
TYPE: POU
LOCALE: 0
IEC_LANGUAGE: ST
PLC_TYPE: independent
PROC_TYPE: independent
GROUP: STRINGS
*)
(*@KEY@:DESCRIPTION*)
version 1.2	25. oct 2008
programmer 	hugo
tested by	tobias

to_lower converts a character from uppercase to lowercase
(*@KEY@:END_DESCRIPTION*)
FUNCTION TO_LOWER:BYTE

(*Group:Default*)

VAR_INPUT
	IN :	BYTE;
END_VAR

(*@KEY@: WORKSHEET
NAME: TO_LOWER
IEC_LANGUAGE: ST
*)
IF in > BYTE#64 AND in < BYTE#91 THEN
   TO_LOWER := in OR BYTE#16#20;
ELSIF (in > BYTE#191 AND in < BYTE#223) AND in <> BYTE#215 AND SETUP_EXTENDED_ASCII(FALSE) THEN
   TO_LOWER := in OR BYTE#16#20;
ELSE
   TO_LOWER := in;
END_IF;

(* revision history
hm	6. mar. 2008	rev 1.0
	original version

hm	19. oct. 2008	rev 1.1
	changed setup constants

ks	25. oct. 2008	rev 1.2
	optimized code
*)
(*@KEY@: END_WORKSHEET *)
END_FUNCTION

(* ---- TO_UPPER.ST ---- *)
(*@PROPERTIES_EX@
TYPE: POU
LOCALE: 0
IEC_LANGUAGE: ST
PLC_TYPE: independent
PROC_TYPE: independent
GROUP: STRINGS
*)
(*@KEY@:DESCRIPTION*)
version 1.3	16. jan. 2009
programmer 	hugo
tested by	oscat

to_upper converts a character from lowercase to uppercase
(*@KEY@:END_DESCRIPTION*)
FUNCTION TO_UPPER:BYTE

(*Group:Default*)

VAR_INPUT
	IN :	BYTE;
END_VAR

(*@KEY@: WORKSHEET
NAME: TO_UPPER
IEC_LANGUAGE: ST
*)
IF in > BYTE#96 AND in < BYTE#123 THEN
   TO_UPPER := in AND BYTE#16#DF;
ELSIF in > BYTE#223 AND in <> BYTE#247 AND in <> BYTE#255 AND SETUP_EXTENDED_ASCII(FALSE) THEN
   TO_UPPER := in AND BYTE#16#DF;
ELSE
   TO_UPPER := in;
END_IF;

(* revision history
hm	6. mar. 2008	rev 1.0
	original version

hm	19. oct. 2008	rev 1.1
	changed setup constants

ks	25. oct. 2008	rev 1.2
	optimized code

hm 16. jan 2009	rev 1.3
	corrected an error in module

*)
(*@KEY@: END_WORKSHEET *)
END_FUNCTION

(* ---- TRIANGLE_A.ST ---- *)
(*@PROPERTIES_EX@
TYPE: POU
LOCALE: 0
IEC_LANGUAGE: ST
PLC_TYPE: independent
PROC_TYPE: independent
GROUP: MATHEMATICAL.GEOMETRY
*)
(*@KEY@:DESCRIPTION*)
version 1.2	10. mar. 2009
programmer 	hugo
tested by	tobias

triangle_A calculates the Area of a triangle.
if any input is 0 it will be neglected and the are will be calculated from eiter:
two sides and an angle (s1 and S2 and the angle A1) or 3 sides.

(*@KEY@:END_DESCRIPTION*)
FUNCTION TRIANGLE_A:REAL

(*Group:Default*)

VAR_INPUT
	S1 :	REAL;
	A :	REAL;
	S2 :	REAL;
	S3 :	REAL;
END_VAR

(*@KEY@: WORKSHEET
NAME: TRIANGLE_A
IEC_LANGUAGE: ST
*)
IF A = 0.0 THEN
	TRIANGLE_A := SQRT((s1+s2+S3) * (s1+s2-S3) * (S2+S3-S1) * (S3+S1-S2)) * 0.25;
ELSE
	TRIANGLE_A := S1 * S2 * SIN(RAD(A)) * 0.5;
END_IF;

(* revision histroy
hm	16. oct 2007	rev 1.0
	original version

hm	22. feb 2008	rev 1.1
	improved performance

hm	10. mar. 2009	rev 1.2
	changed syntax of real constants to 0.0

*)
(*@KEY@: END_WORKSHEET *)
END_FUNCTION

(* ---- UTC_TO_LTIME.ST ---- *)
(*@PROPERTIES_EX@
TYPE: POU
LOCALE: 0
IEC_LANGUAGE: ST
PLC_TYPE: independent
PROC_TYPE: independent
GROUP: TIME_DATE
*)
(*@KEY@:DESCRIPTION*)
version 1.9	27. feb. 2009
programmer 	oscat
tested by	oscat

ltime is a real time clock that uses the system rtc as utc time and calculates and given time zone.
the utc time is supplied on the input UTC.
according to the input variable time_zone_offset when the input dst_enable is true,
the dst on and off times are calculated by a formula for any given year and the time is advanced and reset by one hour
at 02:00 and 03:00 for the last sunday of march and last sunday of october.
the code is high performance and the rtc counts every second.
if more then one time zone is needed by the systen the clock can be started many times by placing more then one function block.
(*@KEY@:END_DESCRIPTION*)
FUNCTION UTC_TO_LTIME:UDINT

(*Group:Default*)

VAR_INPUT
	UTC :	UDINT;
	DST_ENABLE :	BOOL;
	TIME_ZONE_OFFSET :	INT;
END_VAR

VAR
	tmp :	INT;
END_VAR

(*@KEY@: WORKSHEET
NAME: UTC_TO_LTIME
IEC_LANGUAGE: ST
*)
UTC_TO_LTIME := UTC + _INT_TO_UDINT(TIME_ZONE_OFFSET) * UDINT#60 + BOOL_TO_UDINT(DST_ENABLE AND DST(UTC)) * UDINT#3600;

tmp := TIME_ZONE_OFFSET * 60 + BOOL_TO_INT(DST_ENABLE AND DST(UTC)) * 3600;
IF tmp < 0 THEN
	UTC_TO_LTIME := UTC - _INT_TO_UDINT(ABS(tmp));
ELSE
	UTC_TO_LTIME := UTC + _INT_TO_UDINT(tmp);
END_IF;

(* revision history

hm 2.10.2006	rev 1.1
	corrected an error where dst would be delayed by 0.1second

hm 17.1.2007	rev 1.2
	added utc input instead of internal sysrtcgettime because this would only work on wago.
	dst_enable would not be checked before dst would be enabled.

hm 18.3.2007	rev 1.3
	changed code, dst would not work during first cycle.

hm 24.10.2007	rev 1.4
	changed code because the execution every 100ms can cause major problems if the supplied time was not correct at start.
	use of new dst function

hm 12. nov 2007	rev 1.5
		changed Type of time_zone_offset from time to int to allow for time zones with negative offset

hm	8 dec 2007		rev 1.6
	corrected a problem with time_zone_offset

hm	14. oct. 2008	rev 1.7
	renamed module from LTIME to UTC_TO_LTIME
	changed function weekday to day_of_week
	optimized code for better performance

hm	20. oct. 2008	rev 1.8
	changes type of input TIME_ZONE_OFFSET from real to int, now is in +/-minutes
	deleted outputs DST_ON and WDAY
	converted to function

hm	27. feb. 2009	rev 1.9
	added type conversions to avoid warnings under codesys 3.0

*)
(*@KEY@: END_WORKSHEET *)
END_FUNCTION

(* ---- WINDOW.ST ---- *)
(*@PROPERTIES_EX@
TYPE: POU
LOCALE: 0
IEC_LANGUAGE: ST
PLC_TYPE: independent
PROC_TYPE: independent
GROUP: MATHEMATICAL.MATHE
*)
(*@KEY@:DESCRIPTION*)
	version 1.1	22 jan 2007
	programmer 	hugo
	tested BY	tobias

this checks a signal if the signal is between the upper and lower limit
(*@KEY@:END_DESCRIPTION*)
FUNCTION WINDOW:BOOL

(*Group:Default*)

VAR_INPUT
	LOW :	REAL;
	IN :	REAL;
	HIGH :	REAL;
END_VAR

(*@KEY@: WORKSHEET
NAME: WINDOW
IEC_LANGUAGE: ST
*)
window := (in < high) AND (in > low);

(* revision history
hm	22.1.2007	rev 1.1
	changed the order of inputs to low, in, high

*)
(*@KEY@: END_WORKSHEET *)
END_FUNCTION

(* ---- WINDOW2.ST ---- *)
(*@PROPERTIES_EX@
TYPE: POU
LOCALE: 0
IEC_LANGUAGE: ST
PLC_TYPE: independent
PROC_TYPE: independent
GROUP: MATHEMATICAL.MATHE
*)
(*@KEY@:DESCRIPTION*)
	version 1.0	31 oct 2007
	programmer 	hugo
	tested BY	tobias

this checks a signal if the signal is between the upper and lower limit including the two limits
(*@KEY@:END_DESCRIPTION*)
FUNCTION WINDOW2:BOOL

(*Group:Default*)

VAR_INPUT
	LOW :	REAL;
	IN :	REAL;
	HIGH :	REAL;
END_VAR

(*@KEY@: WORKSHEET
NAME: WINDOW2
IEC_LANGUAGE: ST
*)
window2 := (in <= high) AND (in >= low);

(* revision history
hm	31.10.2007	rev 1.0
	original version

*)
(*@KEY@: END_WORKSHEET *)
END_FUNCTION

(* ---- WORD_OF_BYTE.ST ---- *)
(*@PROPERTIES_EX@
TYPE: POU
LOCALE: 0
IEC_LANGUAGE: ST
PLC_TYPE: independent
PROC_TYPE: independent
GROUP: LOGIC.GATE_LOGIC
*)
(*@KEY@:DESCRIPTION*)
version 1.4	18. jul. 2009
programmer 	hugo
tested by	tobias

this function creates a word from 2 individual bytes
(*@KEY@:END_DESCRIPTION*)
FUNCTION WORD_OF_BYTE:WORD

(*Group:Default*)

VAR_INPUT
	B1 :	BYTE;
	B0 :	BYTE;
END_VAR

(*@KEY@: WORKSHEET
NAME: WORD_OF_BYTE
IEC_LANGUAGE: ST
*)
WORD_OF_BYTE := SHL_WORD(BYTE_TO_WORD(B1),8) OR BYTE_TO_WORD(B0);

(* revision history
hm	24. jan 2007	rev 1.0
	original version

hm	2. jan 2008	rev 1.1
	improved performance

hm	19. feb 2008	rev 1.2
	replaced and with or for better compatibility

hm	23. apr. 2008	rev 1.3
	reverse order of inputs to be more logical

hm	18. jul. 2009	rev 1.4
	added type conversions for compatibility reasons

*)
(*@KEY@: END_WORKSHEET *)
END_FUNCTION

(* ---- WORD_OF_DWORD.ST ---- *)
(*@PROPERTIES_EX@
TYPE: POU
LOCALE: 0
IEC_LANGUAGE: ST
PLC_TYPE: independent
PROC_TYPE: independent
GROUP: LOGIC.GATE_LOGIC
*)
(*@KEY@:DESCRIPTION*)
version 1.2	30. oct. 2008
programmer 	hugo
tested by	oscat

this function extracts a single word from the nth position from right (right is lowest byte)
the lower word (starting with Bit0 from in) is selected with N=0.
(*@KEY@:END_DESCRIPTION*)
FUNCTION WORD_OF_DWORD:WORD

(*Group:Default*)

VAR_INPUT
	IN :	DWORD;
	N :	BYTE;
END_VAR

(*@KEY@: WORKSHEET
NAME: WORD_OF_DWORD
IEC_LANGUAGE: ST
*)
WORD_OF_DWORD := DWORD_TO_WORD(SHR(in,_BYTE_TO_INT(SHL(n,4))));

(* revision history
hm	17. jan 2007	rev 1.0
	original version

hm	2. jan 2008		rev 1.1
	improved performance

hm	30. oct. 2008	rev 1.2
	improved performance
*)
(*@KEY@: END_WORKSHEET *)
END_FUNCTION

(* ---- WORD_TO_RANGE.ST ---- *)
(*@PROPERTIES_EX@
TYPE: POU
LOCALE: 0
IEC_LANGUAGE: ST
PLC_TYPE: independent
PROC_TYPE: independent
GROUP: ENGINEERING.SIGNAL_PROCESSING
*)
(*@KEY@:DESCRIPTION*)
version 1.1	10. mar. 2009
programmer 	hugo
tested by	tobias

Word_to_Range converts a Byte into a real between low and high.

(*@KEY@:END_DESCRIPTION*)
FUNCTION WORD_TO_RANGE:REAL

(*Group:Default*)

VAR_INPUT
	X :	WORD;
	LOW :	REAL;
	HIGH :	REAL;
END_VAR

(*@KEY@: WORKSHEET
NAME: WORD_TO_RANGE
IEC_LANGUAGE: ST
*)
WORD_TO_RANGE := (high - low) * _WORD_TO_REAL(X) * 0.00001525902189669640 + low;

(* revision history
hm	9. jan 2008	rev 1.0
	original version

hm	10. mar. 2009	rev 1.1
	improved code
*)

(*@KEY@: END_WORKSHEET *)
END_FUNCTION

(* ---- WORK_WEEK.ST ---- *)
(*@PROPERTIES_EX@
TYPE: POU
LOCALE: 0
IEC_LANGUAGE: ST
PLC_TYPE: independent
PROC_TYPE: independent
GROUP: TIME_DATE
*)
(*@KEY@:DESCRIPTION*)
version 1.5	25. oct. 2008
programmer 	hugo
tested by	oscat

calculates the work week for a given date according to iso8601
(*@KEY@:END_DESCRIPTION*)
FUNCTION WORK_WEEK:INT

(*Group:Parameter*)

VAR_INPUT
	IDATE :	UDINT;
END_VAR

VAR
	d1 :	UDINT;
	w1 :	INT;
	ds :	UDINT;
	yr :	INT;
	w31 :	INT;
	w01 :	INT;
	wm :	INT;
END_VAR

(*@KEY@: WORKSHEET
NAME: WORK_WEEK
IEC_LANGUAGE: ST
*)
(* berechne den 1.1 des jahres von idate. *)
yr := YEAR_OF_DATE(idate);
d1 := year_begin(yr);
(* wochentag von d1 *)
w1 := DAY_OF_WEEK(d1);
(* offset des montags der eletzten KW des vorjahres *)
(* wenn der erste tag des jahres größer als donnerstag ist dann beginnt die letzte kw am montag davor *)
(* wenn der erste tag des jahres ein donnerstag oder kleiner ist beginnt die erste kw 2 montage davor *)
IF w1 < 5 THEN
	ds := d1 - _INT_TO_UDINT(w1+6) * UDINT#86400;
ELSE
	ds := d1 + _INT_TO_UDINT(1-w1) * UDINT#86400;
END_IF;

(* kalenderwoche des eingangsdatums *)
work_week := UDINT_TO_INT((idate - ds) / UDINT#604800);

(* korrektur wenn work_week = 0 *)
IF work_week = 0 THEN
	(* work_week needs to be 53 when 1.jan of the year before is thursday or dec 31. is thursday. *)
	(* first and last weekday of a year is equal and one more day for a leap_year. *)
	IF w1 > 1 THEN w31 := w1 - 1; ELSE W31 := 7; END_IF;
	IF leap_year(yr - 1) THEN IF w31 > 1 THEN w01 := W31 - 1; ELSE w1 := 7; END_IF; END_IF;
	(* if first or last day of a year is a thursday, the year has 53 weeks *)
	WORK_WEEK := 52 + BOOL_TO_INT(w31 = 4 OR w01 = 4);
ELSE
	(* end of year calculation *)
	(* calculated the first and last weekday *)
	IF leap_year(yr) THEN
		IF w1 < 7 THEN w31 := w1 + 1; ELSE w31 := 1; END_IF;
	ELSE
		w31 := w1;
	END_IF;
	(* if first or last day is thursday then the year has 53 weeks otherwise only 52 *)
	wm := 52 + BOOL_TO_INT(w31 = 4 OR w1 = 4);
	IF work_week > wm THEN work_week := 1; END_IF;
END_IF;

(* old code before rev 1.2
w1 := weekday(set_Date(year(idate), 1,1));
IF w1 < 5 THEN
	work_week := (day_of_year(idate) + w1 + 5)/7;
ELSE
	work_week := (day_of_year(idate) + w1 - 2)/7;
END_IF
*)

(* revision history

hm 	17.1.2007		rev 1.1
	deleted unused variable yday

hm	19. dec 2007	rev 1.2
	changed code for better performance
	changed code to comply with ISO8601

hm	16. mar 2008	rev 1.3
	added type conversions to avoid warnings under codesys 3.0

hm	7. oct. 2008	rev 1.4
	changed function year to year_of_date
	changed function weekday to day_of_week

hm	25. oct. 2008	rev 1.5
	optimized code for performance
*)
(*@KEY@: END_WORKSHEET *)
END_FUNCTION

(* ---- YEAR_BEGIN.ST ---- *)
(*@PROPERTIES_EX@
TYPE: POU
LOCALE: 0
IEC_LANGUAGE: ST
PLC_TYPE: independent
PROC_TYPE: independent
GROUP: TIME_DATE
*)
(*@KEY@:DESCRIPTION*)
version 1.2	7. Apr. 2008
programmer 	hugo
tested by	tobias

returs the date of january 1st for the given year
the function works for dates from 1970 - 2099
(*@KEY@:END_DESCRIPTION*)
FUNCTION YEAR_BEGIN:UDINT

(*Group:Default*)

VAR_INPUT
	Y :	INT;
END_VAR

(*@KEY@: WORKSHEET
NAME: YEAR_BEGIN
IEC_LANGUAGE: ST
*)
year_begin := DWORD_TO_UDINT(SHR(UDINT_TO_DWORD(_INT_TO_UDINT(y) * UDINT#1461 - UDINT#2878169),2))  *  UDINT#86400;

(* revision history
hm	19. dec 2007	rev 1.0
	original version

hm	4. jan 2008		rev 1.1
	formula for step7 was incorrect during leap years

hm	7. apr. 2008	rev 1.2
	deleted unused step7 code
*)
(*@KEY@: END_WORKSHEET *)
END_FUNCTION

(* ---- YEAR_END.ST ---- *)
(*@PROPERTIES_EX@
TYPE: POU
LOCALE: 0
IEC_LANGUAGE: ST
PLC_TYPE: independent
PROC_TYPE: independent
GROUP: TIME_DATE
*)
(*@KEY@:DESCRIPTION*)
version 1.1	24. jan. 2011
programmer 	hugo
tested by	oscat

returs the date of december 31st for the given year
the function works for dates from 1970 - 2099

(*@KEY@:END_DESCRIPTION*)
FUNCTION YEAR_END:UDINT

(*Group:Default*)

VAR_INPUT
	Y :	INT;
END_VAR

(*@KEY@: WORKSHEET
NAME: YEAR_END
IEC_LANGUAGE: ST
*)
YEAR_END := DWORD_TO_UDINT(SHR(UDINT_TO_DWORD(INT_TO_UDINT(y) * UDINT#1461 - UDINT#2876712), 2)) * UDINT#86400;

(* revision history
hm	15. jun. 2008	rev 1.0
	original version

hm	24. jan 2011	rev 1.1
	improved performance
*)

(*@KEY@: END_WORKSHEET *)
END_FUNCTION

(* ---- YEAR_OF_DATE.ST ---- *)
(*@PROPERTIES_EX@
TYPE: POU
LOCALE: 0
IEC_LANGUAGE: ST
PLC_TYPE: independent
PROC_TYPE: independent
GROUP: TIME_DATE
*)
(*@KEY@:DESCRIPTION*)
version 1.4	7. oct. 2008
programmer 	hugo
tested by	oscat

returs the year of a date
the function works for dates from 1970 - 2099
(*@KEY@:END_DESCRIPTION*)
FUNCTION YEAR_OF_DATE:INT

(*Group:Default*)

VAR_INPUT
	IDATE :	UDINT;
END_VAR

(*@KEY@: WORKSHEET
NAME: YEAR_OF_DATE
IEC_LANGUAGE: ST
*)
YEAR_OF_DATE := UDINT_TO_INT((idate+UDINT#43200) / UDINT#31557600 + UDINT#1970);

(* code used prior to rev 1.1
year := DWORD_TO_INT((DATE_TO_DWORD(idate)/864+71954300)/36525);
*)

(* revision history
hm	4. aug 2006		rev 1.0
	original version

hm	1. okt 2007		rev 1.1
	corrected error in algorithm
	adjustment for S7 compatibility

hm	23.12.2007		rev 1.2
	changed code for better performance

hm	7. apr. 2008	rev 1.3
	deleted unused step7 code

hm	7. oct. 2008	rev 1.4
	reneamed function (year) to year_of_date

*)
(*@KEY@: END_WORKSHEET *)
END_FUNCTION
